(* CoDeSys 2.3 export: DACHA.EXP *)
(* Libraries: COMlibV2.lb6 25.2.14 08:37:08, ModbusRTU.lib 13.5.15 12:38:16, standard.lib 5.6.98 14:03:02, TcBABasic.lib 22.7.15 15:46:14, TcBase.lib 14.5.09 14:14:08, TcControllerToolbox.lib 19.6.15 13:33:48, TcFloatPC.lib 19.10.09 11:19:54, TcIoFunctions.lib 29.9.20 15:31:50, TcpIp.lib 6.5.15 09:25:52, TcSystem.lib 7.6.16 10:01:22, TcUtilities.lib 3.2.16 15:08:58 *)

(* Task configuration *)
TASK Standard (PRIORITY := 0, INTERVAL := T#2ms);
MAIN();
END_TASK
TASK main2 (PRIORITY := 1, INTERVAL := T#10ms);
MAIN2();
END_TASK

(* Global variable list: Global_Variables *)
VAR_GLOBAL


	Clear						: ClearComBuffer;
	MB							: ModbusRtuMaster_KL6x22B;
	TxBufferCom1				: ComBuffer;
	RxBufferCom1				: ComBuffer;
	SerialLineControlCom1			: SerialLineControl;
	ReceiveDataCom1			: ReceiveData;
	SendDataCom1				: SendData;


	Clear2						: ClearComBuffer;
	MB2							: ModbusRtuMaster_KL6x5B;
	TxBufferCom2				: ComBuffer;
	RxBufferCom2				: ComBuffer;
	SerialLineControlCom2			: SerialLineControl;
	ReceiveDataCom2			: ReceiveData;
	SendDataCom2				: SendData;
(*
	Clear3						: ClearComBuffer;
	MB3							: ModbusRtuMaster_KL6x22B;
	TxBufferCom3				: ComBuffer;
	RxBufferCom3				: ComBuffer;
	SerialLineControlCom3			: SerialLineControl;
	ReceiveDataCom3			: ReceiveData;
	SendDataCom3				: SendData;
*)

	Merc_address				: BYTE:=97;
	Sensor_CO2_high	 			: BYTE;	(*Старший байт датчика MH-Z19B*)
	Sensor_CO2_low 				: BYTE;	(*Младший байт датчика MH-Z19B*)
	iobroker						: iobroker_Struct;
	Modbus						: Modbus_Struct;
	Internal						: Internal_Struct;
	pwm_par_1f,pwm_par_2f		: ST_CTRL_PWM_OUT_PARAMS; (* настройки регулятора*)
	pwm_par_balkon				: ST_CTRL_PWM_OUT_PARAMS; (* настройки регулятора*)
	pwm_par_septik				: ST_CTRL_PWM_OUT_PARAMS; (* настройки регулятора*)
	pwm_par_sauna				: ST_CTRL_PWM_OUT_PARAMS; (* настройки регулятора*)
	pwm_par_fertA				: ST_CTRL_PWM_OUT_PARAMS; (* настройки регулятора*)
	pwm_par_fertB				: ST_CTRL_PWM_OUT_PARAMS; (* настройки регулятора*)

	pi_par_1f						: ST_CTRL_PI_PARAMS;			(*     *)
	pi_par_sauna					: ST_CTRL_PI_PARAMS;			(*     *)
	pi_par_fertA					: ST_CTRL_PI_PARAMS;			(*     *)
	pi_par_fertB					: ST_CTRL_PI_PARAMS;			(*     *)
	pi_par_balkon				: ST_CTRL_PI_PARAMS;			(*     *)

	Timer1					: TON;
	TimerRS485_2			: TON;
	TimerRS485_2Q			 :BOOL;

	TimerRS485_3			: TON;
	TimerRS485_3Q			 :BOOL;

	Timer1Q					: BOOL;
	Timer_day				:TON;
	Timer_dayQ				:BOOL;
	Timer_CO2				:TON;
(*	Timer_CO2Q				:BOOL; *)

	tmCheck					:TON;
	tmCheckQ				: BOOL;

	tmCheckE				:TON;
	tmCheckEQ				: BOOL;

	tmCheckM: TON;
(*
	MB_vars						: stMB;
	Mercury						: stMercury;
	iob_mqtt						: stIobroker;
*)
(*	Sensor_street_north_temp		: REAL;
	Sensor_sport_underfloor_temp	: REAL;
*)
	Sensor_control_temp			: WORD;
	Sensor_control_hum			: WORD;
(*	fert_pwm_levelA	: INT;
	fert_pwm_levelB	: INT;
*)
	Trigger_water_impulse_ponics	: F_TRIG;
	Trigger_A_impulse_ponics		: F_TRIG;
	Trigger_B_impulse_ponics		: F_TRIG;
	Trigger_water_impulse_teplica	: F_TRIG;
	Trigger_fertA_impulse_teplica	: F_TRIG;
	Trigger_fertB_impulse_teplica	: F_TRIG;
	Trigger_water_cnt_impulse_teplica	: F_TRIG;
	Poliv_liters				:	REAL;

	HW_teplica_pomp_fert_level			AT %Q*:BOOL;


(*Terminal 2*)
	HW_heat_first_floor					AT %QX0.0:BOOL;		(* Отопление 1 этаж *)
	HW_heat_second_floor				AT %QX0.1:BOOL;		(* Отопление 2 этаж *)
	HW_heat_sport						AT %QX0.2:BOOL;		(* Отопление спортзал *)
	HW_heat_underfloor					AT %QX0.3:BOOL;		(* Отопление подпол *)
	HW_heat_sauna						AT %QX0.4:BOOL;		(* Отопление сауна *)
	HW_heat_bathroom					AT %QX0.5:BOOL;		(* Отопление душевая *)
	HW_alarm							AT %QX0.6:BOOL;		(* Сирена *)
	HW_power_smoke_sen				AT %QX0.7:BOOL:=FALSE;		(* Питание датчиков дыма *)

(*Terminal 3*)
	HW_vorota							AT %QX1.0:BOOL;		(* Ворота *)
	HW_kalitka							AT %QX1.1:BOOL;		(* Калитка *)
	HW_pomp_house						AT %QX1.2:BOOL;		(* Насос водоснабжения дома *)
	HW_pomp_Garden					AT %QX1.3:BOOL;		(* Свободен*)
	HW_light_garden						AT %QX1.4:BOOL;		(* Прожектор двор *)
	HW_light_rassada						AT %QX1.5:BOOL;		(*Подсветка рассады на балконе *)
	HW_light_rezerv						AT %QX1.6:BOOL;		(* Резервное освещение *)
(*	HW_rezerv_term3_8					AT %QX1.7:BOOL; *)		(* Подогрев трубы в клубнике *)
	HW_poliv_flowers						AT %QX1.7:BOOL;

(*Terminal 4*)
	HW_vent_valve_input					AT %QX2.0:BOOL;		(* Клапан приточной вентиляции и Клапан вытяжной вентиляции *)
	HW_rezerv_term_4_3					AT %QX2.1:BOOL;		(*Свободен*)
	HW_trans_power						AT %QX2.2:BOOL;		(*Подача тока на трансформатор и реле ТЭН-а *)
	HW_vent_in_heat						AT %QX2.3:BOOL;		(* Подогрев притока - ТЭН *)
	HW_valve_pomp_teplica				AT %QX2.4:BOOL;		(* Клапан подачи воды в бочку теплицы*)
	HW_vent_in_trans_105_130				AT %QX2.5:BOOL:=FALSE;  (* Напряжение 110 или 130 В *)
	HW_vent_in_trans_160_220				AT %QX2.6:BOOL:=FALSE;  (* Напряжение 160 или 220 В *)
	HW_vent_in_trans_LO_HI				AT %QX2.7:BOOL:=FALSE;  (* Напряжение 110/130  или 160/220 В *)

(*Terminal 5*)
	HW_poliv_terrasa						AT %QX3.0:BOOL;		(* полив терраса  *)
	HW_poliv_zapad						AT %QX3.1:BOOL;		(* полив запад   *)
	HW_poliv_south						AT %QX3.2:BOOL;		(* полив юг   *)
	HW_poliv_north						AT %QX3.3:BOOL;		(* полив север   *)
	HW_septik_heat						AT %QX3.4:BOOL;		(*подогрев трубы до септика*)
	HW_power_supply_parnik				AT %QX3.5:BOOL;		(* Подача питания для механизма открывания окна*)
	HW_power_polarity_parnik				AT %QX3.6:BOOL;		(* Полярность питания для механизма открывания окна*)
	HW_parnik_heat						AT %QX3.7:BOOL;		(* подогрев трубы в парнике*)

(*Terminal 6*)
	HW_teplica_pomp_poliv				AT %Q*:BOOL; (*Teplica GR1.1*)
	HW_teplica_light						AT %Q*:BOOL; (*Teplica GR1.2*)
	HW_rezerv_6_3						AT %Q*:BOOL; (*Свободен*)
	HW_rezerv_6_4						AT %Q*:BOOL; (*Свободен*)
	HW_rezerv_6_5						AT %Q*:BOOL; (*Свободен*)
	HW_rezerv_6_6						AT %Q*:BOOL; (*Свободен*)
	HW_teplica_vent						AT %Q*:BOOL; (*Teplica GR1.7*)
	HW_teplica_heat						AT %Q*:BOOL; (*Teplica GR1.8*)




(*Terminal 7*)
	HW_rezerv_7_1						AT %Q*:BOOL;
	HW_rezerv_7_2						AT %Q*:BOOL;
	HW_rezerv_7_3						AT %Q*:BOOL;
	HW_ponics_pomp_water				AT %Q*:BOOL; (* 4 *)
	HW_ponics_pomp_tankA				AT %Q*:BOOL; (* 5 *)
	HW_ponics_pomp_tankB				AT %Q*:BOOL; (* 6 *)
	HW_ponics_pomp_main				AT %Q*:BOOL; (* 7 *)
	HW_balkon_heat						AT %Q*:BOOL; (* 8 *)

(*Terminal 8*)

(*	HW_teplica_pomp_fertA				AT %Q*:BOOL; (* PWM GND fert A*) (*Teplica GR2.1*)
	HW_teplica_pomp_fertB				AT %Q*:BOOL; (* PWM GND fert B*) (*Teplica GR2.2*)
*)
	fert_pwm_levelA						AT %Q*: UINT;
	fert_pwm_levelB						AT %Q*: UINT;
	pwm_ctrl_1							AT %Q*: USINT;
	pwm_ctrl_2							AT %Q*: USINT;


(*Terminal 9*)

	HW_PIR_terrasa						AT %IX56.0:BOOL;		(*PIR датчик терраса *)
	HW_PIR_zapad						AT %IX56.1:BOOL;		(*PIR датчик запад *)
	HW_PIR_vostok						AT %IX56.2:BOOL;		(*PIR датчик восток *)
	HW_PIR_sport						AT %IX56.3:BOOL;		(*PIR датчик спортзал *)
	HW_GERKON_drovnik					AT %IX56.4:BOOL;		(*Геркон дровник *)
	HW_GERKON_door					AT %IX56.5:BOOL;		(*Геркон дверь *)
	HW_sensor_smoke_1floor				AT %IX56.6:BOOL;		(*Датчик дыма 1 этаж *)
	HW_sensor_smoke_2floor				AT %IX56.7:BOOL;		(*Датчик дыма 2 этаж *)

(*Terminal 10*)
	HW_button_light_garden				AT %IX57.0:BOOL;		(* Кнопка прожектор терраса  *)
	HW_sensor_smoke_sport				AT %IX57.1:BOOL;		(*Датчик дыма спорт *)
	HW_button_vorota						AT %IX57.2:BOOL;		(* Кнопка открытия ворот  *)
	HW_rezerv_term_10_4					AT %IX57.3:BOOL;		(* Кнопка открытия калитки  *)
	HW_button_poliv_terrasa				AT %IX57.4:BOOL;		(* Кнопка полив терраса 2 часа  *)
	HW_button_poliv_zapad				AT %IX57.5:BOOL;		(* Кнопка полив запад  2 часа  *)
	HW_button_poliv_south				AT %IX57.6:BOOL;		(*  Кнопка полив юг  2 часа  *)
	HW_button_poliv_north					AT %IX57.7:BOOL;		(*  Кнопка полив север  2 часа  *)
(*Terminal 11*)
	HW_sensor_supply					AT %IX58.0:BOOL;		(* Датчик напряжения 220В  *)
	HW_GERKON_sklad					AT %IX58.1:BOOL;		(*Геркон склад*)
	HW_PIR_north_zapad					AT %IX58.2:BOOL;		(*PIR датчик  северо-запад*)
	HW_PIR_north_vostok					AT %IX58.3:BOOL;		(*PIR датчик  северо-восток*)

(*Terminal 12*)
	HW_vent_relay_pressure				 AT	%I*	:BOOL;		(*Реле давления вентиляции*)
	HW_sensor_smoke_stair				AT	%I*	:BOOL;		(*Датчик дыма лестница *)
	HW_sensor_smoke_3floor				AT	%I*	:BOOL;		(*Датчик дыма 3 этаж *)
	HW_sensor_smoke_drovnik			AT	%I*	:BOOL;		(*Датчик дыма дровник *)
	HW_sensor_smoke_sklad				AT	%I*	:BOOL;		(*Датчик дыма склад *)
	HW_button_alarm						AT	%I*	:BOOL;		(*Кнопка вкл и откл сирены *)
	HW_battery_low						 AT	%I*	:BOOL;		(*Датик низкого напряжения АКБ *)
	HW_water_tank_teplica_level			 AT	%I*	:BOOL;		(*Датчик уровня воды в бочке в теплице *) (*Teplica GR2.3*)

(*Terminal 13*)
	HW_water_tank_ponics_level_low		 AT	%I*	:BOOL;
	HW_water_tank_ponics_level_high		 AT	%I*	:BOOL;
	HW_sensor_fluid_alarm				 AT	%I*	:BOOL;
	HW_water_counter					 AT	%I*	:BOOL;
	HW_I_rez5							 AT	%I*	:BOOL;
	HW_I_rez6							 AT	%I*	:BOOL;
	HW_I_rez7							 AT	%I*	:BOOL;
	HW_I_rez8							 AT	%I*	:BOOL;

(*Terminal 14*)
	HW_impulse_water_teplica				 AT	%I*	:BOOL; (*Teplica GR2.4*)
	HW_impulse_fertA_teplica				 AT	%I*	:BOOL; (*Teplica GR2.5*)
	HW_impulse_fertB_teplica				 AT	%I*	:BOOL; (*Teplica GR2.6*)
	HW_impulse_water_ponics				 AT	%I*	:BOOL;

	HW_impulse_tankA_ponics				 AT	%I*	:BOOL;
	HW_impulse_tankB_ponics				 AT	%I*	:BOOL;
	HW_I_rez15							 AT	%I*	:BOOL;
	HW_I_rez16							 AT	%I*	:BOOL;

(*Terminal 15*)
	HW_temp_first_floor					AT %IW40:INT;	(* Датчик температуры 1 этаж *)
	HW_temp_second_floor				AT %IW42:INT;	(* Датчик температуры 2 этаж *)
	HW_temp_sauna						AT %IW44:INT;	(* Датчик температуры сауна*)
	HW_temp_sport						AT %IW46:INT;	(* Датчик температуры спортзал *)

(*Terminal 16*)
	HW_temp_underfloor					AT %IW48:INT;	(* Датчик температуры подпол *)
	HW_temp_balkon						AT %IW50:INT;	(* Датчик температуры  *)
	HW_temp_street						AT %IW52:INT;	(* Датчик температуры улица *)
	HW_temp_vent						AT %IW54:INT;	(* Датчик температуры притока вентиляции *)



END_VAR

(* Global variable list: TwinCAT_Configuration *)
(* Generated automatically by TwinCAT - (read only) *)
VAR_CONFIG
	MAIN2.ToFromNovRam AT %QB584 : DataToFromNovram;	(*  ~ {LinkedWith:TIID^Device 2 (NOV/DP-RAM)^Outputs^Var 403} *)
	.MB.InData AT %IB68 : MB_KL6inData22B;
	.MB.OutData AT %QB376 : MB_KL6outData22B;
	.MB2.InData AT %IB96 : MB_KL6inData5B;
	.MB2.OutData AT %QB344 : MB_KL6outData5B;
	.HW_teplica_pomp_fert_level AT %QX476.0 : BOOL;
	.HW_teplica_pomp_poliv AT %QX480.3 : BOOL;	(*  ~ {LinkedWith:TIID^Device 1 (CX9000-KBus)^CX9000-KB^Term 6 (KL2408)^Channel 1^Output} *)
	.HW_teplica_light AT %QX480.2 : BOOL;	(*  ~ {LinkedWith:TIID^Device 1 (CX9000-KBus)^CX9000-KB^Term 6 (KL2408)^Channel 2^Output} *)
	.HW_rezerv_6_3 AT %QX724.0 : BOOL;	(*  ~ {LinkedWith:TIID^Device 1 (CX9000-KBus)^CX9000-KB^Term 6 (KL2408)^Channel 3^Output} *)
	.HW_rezerv_6_4 AT %QX724.1 : BOOL;	(*  ~ {LinkedWith:TIID^Device 1 (CX9000-KBus)^CX9000-KB^Term 6 (KL2408)^Channel 4^Output} *)
	.HW_rezerv_6_5 AT %QX724.2 : BOOL;	(*  ~ {LinkedWith:TIID^Device 1 (CX9000-KBus)^CX9000-KB^Term 6 (KL2408)^Channel 5^Output} *)
	.HW_rezerv_6_6 AT %QX724.3 : BOOL;	(*  ~ {LinkedWith:TIID^Device 1 (CX9000-KBus)^CX9000-KB^Term 6 (KL2408)^Channel 6^Output} *)
	.HW_teplica_vent AT %QX480.0 : BOOL;	(*  ~ {LinkedWith:TIID^Device 1 (CX9000-KBus)^CX9000-KB^Term 6 (KL2408)^Channel 7^Output} *)
	.HW_teplica_heat AT %QX480.1 : BOOL;	(*  ~ {LinkedWith:TIID^Device 1 (CX9000-KBus)^CX9000-KB^Term 6 (KL2408)^Channel 8^Output} *)
	.HW_rezerv_7_1 AT %QX724.4 : BOOL;	(*  ~ {LinkedWith:TIID^Device 1 (CX9000-KBus)^CX9000-KB^Term 7 (KL2408)^Channel 1^Output} *)
	.HW_rezerv_7_2 AT %QX724.5 : BOOL;	(*  ~ {LinkedWith:TIID^Device 1 (CX9000-KBus)^CX9000-KB^Term 7 (KL2408)^Channel 2^Output} *)
	.HW_rezerv_7_3 AT %QX724.6 : BOOL;	(*  ~ {LinkedWith:TIID^Device 1 (CX9000-KBus)^CX9000-KB^Term 7 (KL2408)^Channel 3^Output} *)
	.HW_ponics_pomp_water AT %QX484.2 : BOOL;	(*  ~ {LinkedWith:TIID^Device 1 (CX9000-KBus)^CX9000-KB^Term 7 (KL2408)^Channel 4^Output} *)
	.HW_ponics_pomp_tankA AT %QX484.3 : BOOL;	(*  ~ {LinkedWith:TIID^Device 1 (CX9000-KBus)^CX9000-KB^Term 7 (KL2408)^Channel 5^Output} *)
	.HW_ponics_pomp_tankB AT %QX484.4 : BOOL;	(*  ~ {LinkedWith:TIID^Device 1 (CX9000-KBus)^CX9000-KB^Term 7 (KL2408)^Channel 6^Output} *)
	.HW_ponics_pomp_main AT %QX484.1 : BOOL;	(*  ~ {LinkedWith:TIID^Device 1 (CX9000-KBus)^CX9000-KB^Term 7 (KL2408)^Channel 7^Output} *)
	.HW_balkon_heat AT %QX580.0 : BOOL;	(*  ~ {LinkedWith:TIID^Device 1 (CX9000-KBus)^CX9000-KB^Term 7 (KL2408)^Channel 8^Output} *)
	.fert_pwm_levelA AT %QB708 : UINT;	(*  ~ {LinkedWith:TIID^Device 1 (CX9000-KBus)^CX9000-KB^Term 8 (KL2502)^Channel 1^Data Out} *)
	.fert_pwm_levelB AT %QB710 : UINT;	(*  ~ {LinkedWith:TIID^Device 1 (CX9000-KBus)^CX9000-KB^Term 8 (KL2502)^Channel 2^Data Out} *)
	.pwm_ctrl_1 AT %QB712 : USINT;	(*  ~ {LinkedWith:TIID^Device 1 (CX9000-KBus)^CX9000-KB^Term 8 (KL2502)^Channel 1^Ctrl} *)
	.pwm_ctrl_2 AT %QB713 : USINT;	(*  ~ {LinkedWith:TIID^Device 1 (CX9000-KBus)^CX9000-KB^Term 8 (KL2502)^Channel 2^Ctrl} *)
	.HW_vent_relay_pressure AT %IX104.0 : BOOL;	(*  ~ {LinkedWith:TIID^Device 1 (CX9000-KBus)^CX9000-KB^Term 12 (KL1408)^Channel 1^Input} *)
	.HW_sensor_smoke_stair AT %IX140.0 : BOOL;	(*  ~ {LinkedWith:TIID^Device 1 (CX9000-KBus)^CX9000-KB^Term 12 (KL1408)^Channel 2^Input} *)
	.HW_sensor_smoke_3floor AT %IX132.1 : BOOL;	(*  ~ {LinkedWith:TIID^Device 1 (CX9000-KBus)^CX9000-KB^Term 12 (KL1408)^Channel 3^Input} *)
	.HW_sensor_smoke_drovnik AT %IX132.2 : BOOL;	(*  ~ {LinkedWith:TIID^Device 1 (CX9000-KBus)^CX9000-KB^Term 12 (KL1408)^Channel 4^Input} *)
	.HW_sensor_smoke_sklad AT %IX132.3 : BOOL;	(*  ~ {LinkedWith:TIID^Device 1 (CX9000-KBus)^CX9000-KB^Term 12 (KL1408)^Channel 5^Input} *)
	.HW_button_alarm AT %IX136.0 : BOOL;	(*  ~ {LinkedWith:TIID^Device 1 (CX9000-KBus)^CX9000-KB^Term 12 (KL1408)^Channel 6^Input} *)
	.HW_battery_low AT %IX132.0 : BOOL;	(*  ~ {LinkedWith:TIID^Device 1 (CX9000-KBus)^CX9000-KB^Term 12 (KL1408)^Channel 7^Input} *)
	.HW_water_tank_teplica_level AT %IX144.0 : BOOL;	(*  ~ {LinkedWith:TIID^Device 1 (CX9000-KBus)^CX9000-KB^Term 12 (KL1408)^Channel 8^Input} *)
	.HW_water_tank_ponics_level_low AT %IX168.0 : BOOL;	(*  ~ {LinkedWith:TIID^Device 1 (CX9000-KBus)^CX9000-KB^Term 13 (KL1408)^Channel 1^Input} *)
	.HW_water_tank_ponics_level_high AT %IX168.1 : BOOL;	(*  ~ {LinkedWith:TIID^Device 1 (CX9000-KBus)^CX9000-KB^Term 13 (KL1408)^Channel 2^Input} *)
	.HW_sensor_fluid_alarm AT %IX164.0 : BOOL;	(*  ~ {LinkedWith:TIID^Device 1 (CX9000-KBus)^CX9000-KB^Term 13 (KL1408)^Channel 3^Input} *)
	.HW_water_counter AT %IX164.1 : BOOL;	(*  ~ {LinkedWith:TIID^Device 1 (CX9000-KBus)^CX9000-KB^Term 13 (KL1408)^Channel 4^Input} *)
	.HW_I_rez5 AT %IX148.4 : BOOL;	(*  ~ {LinkedWith:TIID^Device 1 (CX9000-KBus)^CX9000-KB^Term 13 (KL1408)^Channel 5^Input} *)
	.HW_I_rez6 AT %IX148.5 : BOOL;	(*  ~ {LinkedWith:TIID^Device 1 (CX9000-KBus)^CX9000-KB^Term 13 (KL1408)^Channel 6^Input} *)
	.HW_I_rez7 AT %IX148.6 : BOOL;	(*  ~ {LinkedWith:TIID^Device 1 (CX9000-KBus)^CX9000-KB^Term 13 (KL1408)^Channel 7^Input} *)
	.HW_I_rez8 AT %IX148.7 : BOOL;	(*  ~ {LinkedWith:TIID^Device 1 (CX9000-KBus)^CX9000-KB^Term 13 (KL1408)^Channel 8^Input} *)
	.HW_impulse_water_teplica AT %IX152.0 : BOOL;	(*  ~ {LinkedWith:TIID^Device 1 (CX9000-KBus)^CX9000-KB^Term 14 (KL1408)^Channel 1^Input} *)
	.HW_impulse_fertA_teplica AT %IX152.1 : BOOL;	(*  ~ {LinkedWith:TIID^Device 1 (CX9000-KBus)^CX9000-KB^Term 14 (KL1408)^Channel 2^Input} *)
	.HW_impulse_fertB_teplica AT %IX152.2 : BOOL;	(*  ~ {LinkedWith:TIID^Device 1 (CX9000-KBus)^CX9000-KB^Term 14 (KL1408)^Channel 3^Input} *)
	.HW_impulse_water_ponics AT %IX156.0 : BOOL;	(*  ~ {LinkedWith:TIID^Device 1 (CX9000-KBus)^CX9000-KB^Term 14 (KL1408)^Channel 4^Input} *)
	.HW_impulse_tankA_ponics AT %IX156.1 : BOOL;	(*  ~ {LinkedWith:TIID^Device 1 (CX9000-KBus)^CX9000-KB^Term 14 (KL1408)^Channel 5^Input} *)
	.HW_impulse_tankB_ponics AT %IX156.2 : BOOL;	(*  ~ {LinkedWith:TIID^Device 1 (CX9000-KBus)^CX9000-KB^Term 14 (KL1408)^Channel 6^Input} *)
	.HW_I_rez15 AT %IX149.6 : BOOL;	(*  ~ {LinkedWith:TIID^Device 1 (CX9000-KBus)^CX9000-KB^Term 14 (KL1408)^Channel 7^Input} *)
	.HW_I_rez16 AT %IX149.7 : BOOL;	(*  ~ {LinkedWith:TIID^Device 1 (CX9000-KBus)^CX9000-KB^Term 14 (KL1408)^Channel 8^Input} *)
END_VAR

(* Data type *)
TYPE DataToFromNovram :
STRUCT

	Target_CO2_mem					:		INT:=600;
	First_floor_temp_target_mem		:		INT:=5;
	Second_floor_temp_target_mem		:		INT:=5;
	Sport_temp_target_mem			:		INT:=5;
	Sauna_temp_target_mem			:		INT:=5;
	Underfloor_temp_target_mem		:		INT:=5;
	Underfloor_humidity_target_mem	:		INT:=90;

	Pomp_house_mem				:		BOOL:=FALSE;
	Pomp_garden_mem				:		BOOL:=FALSE;

	Light_garden_mem				:		BOOL:=FALSE;

	Vent_mem						:		BOOL:=FALSE;
	Vent_heat_mem					:		INT;
	Vent_heat_level_mem				:		BOOL;

	Poliv_zapad_minutes				:		INT:=90;
	Poliv_terrasa_minutes				:		INT:=90;
	Poliv_south_minutes				:		INT:=90;
	Poliv_north_minutes				:		INT:=90;

	Teplica_temp_set_high			:	INT:=21;
	Teplica_temp_set_low				:	INT:=18;
	Teplica_light_set_low				:	INT:=4000;
	Teplica_light_allow				:	BOOL;
	Teplica_poliv_kf					:	INT:=1025;
	Teplica_fertA_kf					:	INT:=11450;
	Teplica_fertB_kf					:	INT:=11450;

	Teplica_set_poliv					:	REAL;
	Teplica_set_fertA					:	REAL;
	Teplica_set_fertB					:	REAL;
	Teplica_set_max_poliv_time		:	UDINT;
	Teplica_set_max_fertA_time		:	UDINT;
	Teplica_set_max_fertB_time		:	UDINT;
	Teplica_set_clear_time			:	UDINT:=5;

	Teplica_set_temp_pomp_cold		:	INT:=24;
	Teplica_set_temp_window_open	:	INT:=21;
	Teplica_set_poliv_before_fert		:	INT:=50;

	Teplica_set_temp_tank			:	INT:=-60;
	Teplica_fert_kf					:	INT:=12;
	Teplica_zone_poliv				:	BOOL;
	Teplica_type_fert					:	BOOL;
	Teplica_type_poliv				:	BOOL;
	Teplica_set_finish_clear_time		:	INT:=5;
	Teplica_set_finish_clear_vol		:	INT:=1;

	Ponics_start_mintutes_poliv			:	INT:=0;
	Ponics_start_minutes_doliv_AB		:	INT:=30;
	Ponics_start_minutes_doliv_water	:	INT:=20;
	Ponics_set_doliv_AB				:	REAL:=0.1;
	Ponics_set_doliv_water			:	REAL:=3;
	Ponics_set_max_poliv_time			:	INT:=3000;
	Ponics_set_max_doliv_A_time		:	INT:=30;
	Ponics_set_max_doliv_water_time	:	INT:=600;
	Ponics_set_EC					:	REAL:=2.0;
	Balkon_set_temp					:	INT:=21;
	Ponics_A_kf						:	INT:=7030;
	Ponics_B_kf						:	INT:=7030;
	Ponics_water_kf					:	INT:=7030;

	Sensor_house_water_imp			:	UDINT;
	Parnik_temp_step1_window			:	INT:=18;
	Parnik_temp_step2_window			:	INT:=24;
	Parnik_set_auto_window			:	BOOL;
	Parnik_current_level_window		:	INT;
	Parnik_manual_level_window		:	INT;



END_STRUCT
END_TYPE

(* Data type *)
TYPE DataToFromNovram2 :
STRUCT

	Target_CO2_mem					:		INT;
	First_floor_temp_target_mem		:		INT;
	Second_floor_temp_target_mem		:		INT;
	Sport_temp_target_mem			:		INT;
	Sauna_temp_target_mem			:		INT;
	Underfloor_temp_target_mem		:		INT;
	Underfloor_humidity_target_mem	:		INT;

	Pomp_house_mem				:		BOOL;
	Pomp_garden_mem				:		BOOL;

	Light_garden_mem				:		BOOL;

	Vent_mem						:		BOOL;
	Vent_heat_mem					:		INT;
	Vent_heat_level_mem				:		BOOL;

	Poliv_zapad_minutes				:		INT;
	Poliv_terrasa_minutes				:		INT;
	Poliv_south_minutes				:		INT;
	Poliv_north_minutes				:		INT;

	Teplica_temp_set_high			:	INT;
	Teplica_temp_set_low				:	INT;
	Teplica_light_set_low				:	INT;
	Teplica_light_allow				:	BOOL;
	Teplica_poliv_kf					:	INT;
	Teplica_fertA_kf					:	INT;
	Teplica_fertB_kf					:	INT;

	Teplica_set_poliv					:	REAL;
	Teplica_set_fertA					:	REAL;
	Teplica_set_fertB					:	REAL;
	Teplica_set_max_poliv_time		:	UDINT;
	Teplica_set_max_fertA_time		:	UDINT;
	Teplica_set_max_fertB_time		:	UDINT;
	Teplica_set_clear_time			:	UDINT;

END_STRUCT
END_TYPE

(* Data type *)
TYPE Internal_struct :
STRUCT
	Drovnik_temp					 :	REAL; 	(*12382*)			(* PT1000 *)
	Sklad_temp					 :	REAL; 	(*12384*)			(* PT1000 *)
	Rezerv_temp					 :	REAL; 	(*12386*)			(* PT1000 *)

	First_floor_temp 				:	REAL;	(*12288+100=12388*) (* PT1000 *)
	First_floor_hum 				:	REAL;	(*12390*)			(*SHT20		#1*)
	First_floor_CO2				:	REAL;	(*12392*)
	First_floor_temp_SHT30		:	REAL;	(*12394*)			(*SHT20		#1*)

	Second_floor_hum			:	REAL;	(*12396*)			(*SHT20		#2*)
	Second_floor_temp 			:	REAL;	(*12398*) 		(* PT1000 *)
	Second_floor_CO2 			:	REAL;	(*12400*)
	Sport_temp	 				:	REAL;	(*12402*)			(* PT1000 *)

	Sauna_temp	 				:	REAL;	(*12404*)			(* PT1000 *)
	Underfloor_temp				:	REAL;	(*12406*)			(* PT1000 *)
	Underfloor_hum				:	REAL;	(*12408*)			(*SHT20		#3*)
	Sport_underfloor_temp			:	REAL;	(*12410*)			(* PT1000 *)

	Sport_underfloor_hum			:	REAL;	(*12412*)			(*SHT20		#4*)
	Street_temp					:	REAL;	(*12414*)			(* PT1000 *)
	Vent_temp					:	REAL;	(*12416*)			(* PT1000 *)
	Sklad_temp_SHT20			:	REAL;	(*12418*)			(*SHT20		#5*)
	Sklad_hum					:	REAL;	(*12420*)			(*SHT20		#5*)
	Temp_vent_in				:	REAL;	(*12422*)			(* unused *)

	Sport_temp_SHT30			:	REAL;	(*12458 *)		(*SHT20		#6*)
	Sport_hum					:	REAL;	(*12460 *)		(*SHT20		#6*)
	Drovnik_temp_SHT30			:	REAL;	(*12462 *)		(*SHT20		#6*)
	Drovnik_hum					:	REAL;	(*12464 *)		(*SHT20		#6*)


	Uv1							:	REAL;	(*12424*)
	Uv2							:	REAL;	(*12426*)
	Uv3							:	REAL;	(*12428*)
	Pw1							:	REAL;	(*12430*)
	Pw2							:	REAL;	(*12432*)
	Pw3							:	REAL;	(*12434*)
	Pw_total						:	REAL;	(*12436*)
	Ia1							:	REAL;	(*12438*)
	Ia2							:	REAL;	(*12440*)
	Ia3							:	REAL;	(*12442*)
	E_T1						:	REAL;	(*12444*)
	E_T2						:	REAL; 	(*12288+158=12446*)

	Second_floor_temp_SHT30			:	REAL;	(*12448 *)		(*SHT20		#2*)
	Underfloor_temp_SHT30			:	REAL;	(*12450 *)		(*SHT20		#3*)
	Sport_underfloor_temp_SHT30		:	REAL;	(*12452 *)		(*SHT20		#4*)
	Street_temp_SHT20				:	REAL;	(*12454 *)		(*SHT20		#6*)
	Street_hum						:	REAL;	(*12456 *)		(*SHT20		#6*)

	Teplica_temp_SHT30				:	REAL;	(**)
	Teplica_hum_SHT30				:	REAL;	(**)


END_STRUCT
END_TYPE

(* Data type *)
TYPE iobroker_Struct  :
STRUCT
(*	Vent_status				: 	INT;
	Valve_status				: 	INT;
	First_floor_temp 			:	REAL;
	First_floor_temp_target 		:	INT;
	First_floor_hum 			:	REAL;
	First_floor_CO2			:	REAL;
	Kitchen_room_temp		:	REAL;
	Kitchen_room_hum		:	REAL;
	Second_floor_temp 		:	REAL;
	Second_floor_temp_target 	:	INT;
	Second_floor_CO2 		:	REAL;
	Sport_temp	 			:	REAL;
	Sport_temp_target			:	INT;
	Sauna_temp	 			:	REAL;
	Sauna_temp_target		:	INT;
	Underfloor_temp			:	REAL;
	Underfloor_temp_target	:	INT;
	Underfloor_humidity		:	REAL;
	Underfloor_humidity_target	:	INT;
	Sport_underfloor_temp		:	REAL;
	Sport_underfloor_hum		:	REAL;
	Street_temp				:	REAL;
	Vent_temp				:	REAL;
	Street_north_temp			:	REAL;
	Street_north_hum			:	REAL;
*)
	PIR_terrasa				:	BOOL:=TRUE;
	PIR_zapad				:	BOOL:=TRUE;
	PIR_vostok				:	BOOL:=TRUE;
	PIR_sport				:	BOOL:=TRUE;
	GERKON_drovnik			:	BOOL:=TRUE;
	Smoke					:	BOOL;
	Button_light_garden		:	BOOL;
	Light_garden				:	BOOL;
	Vorota_active				:	BOOL:=FALSE;
	Vorota_open_active		:	BOOL:=FALSE;
(*	Poliv_zapad				:	BOOL;
	Poliv_terrasa				:	BOOL;
	Poliv_south				:	BOOL;
	Poliv_north				:	BOOL;
*)
(*
	Vent_input_level			:	INT;  (*  0-220 V  *)
	Vent_output_level			:	INT; (*0-100%*)
	Temp_vent_in			:	REAL;
	Vent_valve_status			:	INT;
	Security_status			:	BOOL;
	Target_CO2				:	INT;
	Vent						:	BOOL;
	Vent_underfloor			:	BOOL;
	Vent_out					:	BOOL;
	Vent_heat				:	INT;
	Vent_heat_level			:	BOOL;
	Vorota					:	BOOL;
	Vorota_open				:	BOOL;
	Kalitka					:	BOOL;
	
	Sensor_supply			:	BOOL;
	Pomp_house				:	BOOL;
	Pomp_garden			:	BOOL;
	Light_garden				:	BOOL;
	Poliv_zapad				:	BOOL;
	Poliv_terrasa				:	BOOL;
	Poliv_south				:	BOOL;
	Poliv_zapad_minutes		:	INT;
	Poliv_terrasa_minutes		:	INT;
	Poliv_south_minutes		:	INT;
	Uv1						:	REAL;
	Uv2						:	REAL;
	Uv3						:	REAL;
	Pw1						:	REAL;
	Pw2						:	REAL;
	Pw3						:	REAL;
	Pw_total					:	REAL;
	Ia1						:	REAL;
	Ia2						:	REAL;
	Ia3						:	REAL;
	E_T1					:	REAL;
	E_T2					:	REAL; (* 64 values*)
*)

(*	M1T1					:	DWORD:=0;
	M1T2					:	DWORD:=0; (* 66 values*)

	M2T1					:	DWORD:=0; (* 67 values*)
	M2T2					:	DWORD:=0;
	M3T1					:	DWORD:=0;
	M3T2					:	DWORD:=0;
	M4T1					:	DWORD:=0; (* 70 values*)
	M4T2					:	DWORD:=0;
	M5T1					:	DWORD:=0;
	M5T2					:	DWORD:=0;
	M6T1					:	DWORD:=0;
	M6T2					:	DWORD:=0;
	M7T1					:	DWORD:=0;
	M7T2					:	DWORD:=0;
	M8T1					:	DWORD:=0;
	M8T2					:	DWORD:=0;
	M9T1					:	DWORD:=0;
	M9T2					:	DWORD:=0;
	M10T1					:	DWORD:=0;
	M10T2					:	DWORD:=0;
	M11T1					:	DWORD:=0;
	M11T2					:	DWORD:=0;
	M12T1					:	DWORD:=0;
	M12T2					:	DWORD:=0;   (* 86 values*)
*)

END_STRUCT
END_TYPE

(* Data type *)
TYPE Modbus_struct :
STRUCT

	M1T1							AT %MW0	:REAL;  	(* modbus address 12288 *)
	M1T2							AT %MW4	:REAL;	(* 12290 *)
	M2T1							AT %MW8	:REAL;	(* 12292 *)
	M2T2							AT %MW12	:REAL;	 (* 12294 *)
	M3T1							AT %MW16	:REAL;	 (* 12296 *)
	M3T2							AT %MW20	:REAL;	 (* 12298 *)
	M4T1							AT %MW24	:REAL;	 (* 12300 *)
	M4T2							AT %MW28	:REAL;	 (* 12302 *)
	M5T1							AT %MW32	:REAL;	 (* 12304 *)
	M5T2							AT %MW36	:REAL;	 (* 12306 *)
	M6T1							AT %MW40	:REAL;	 (* 12308 *)
	M6T2							AT %MW44	:REAL;	(* 12310 *)
	M7T1							AT %MW48	:REAL;	 (* 12312 *)
	M7T2							AT %MW52	:REAL;	 (* 12314 *)
	M8T1							AT %MW56	:REAL;	 (* 12316 *)
	M8T2							AT %MW60	:REAL;	(* 12318 *)
	M9T1							AT %MW64	:REAL;	(* 12320 *)
	M9T2							AT %MW68	:REAL;	(* 12322 *)
	M10T1							AT %MW72	:REAL;	(* 12324 *)
	M10T2							AT %MW76	:REAL;	(* 12326 *)
	M11T1							AT %MW80	:REAL;	(* 12328 *)
	M11T2							AT %MW84	:REAL;	(* 12330 *)
	M12T1							AT %MW88	:REAL;	(* 12332 *)
	M12T2							AT %MW92	:REAL;	(* 12334 *)


	Vent_status					AT %MB100	:	INT;		(*12288+50=12338*)
	Valve_status					AT %MB102	: 	INT;		(*12339*)
	First_floor_temp_target 			AT %MB104	:	INT:=5;		(*12340*)
	Second_floor_temp_target 		AT %MB106	:	INT:=5;		(*12341*)
	Sport_temp_target				AT %MB108	:	INT:=5;		(*12342*)
	Sauna_temp_target			AT %MB110	:	INT:=0;		(*12343*)
	Underfloor_temp_target		AT %MB112	:	INT:=5;		(*12344*)
	Underfloor_humidity_target		AT %MB114	:	INT:=90;		(*12345*)
	PIR_terrasa					AT %MB116	:	BOOL:=TRUE;	(*12346*)
	PIR_zapad					AT %MB118	:	BOOL:=TRUE;	(*12347*)
	PIR_vostok					AT %MB120	:	BOOL:=TRUE;	(*12348*)
	PIR_sport					AT %MB122	:	BOOL:=TRUE;	(*12349*)
	GERKON_drovnik				AT %MB124	:	BOOL:=TRUE;	(*12288+62=12350*)

	Vent_input_level				AT %MB126	:	INT; 			 (*12351			*  0-220 V  *)
	Vent_output_level				AT %MB128	:	INT; 			(*12352			0-100%*)
	Vent_valve_status				AT %MB130	:	INT;		(*12353*)
	Target_CO2					AT %MB132	:	INT:=600;		(*12354*)
	Security_status				AT %MB134	:	BOOL;	(*12355*)
	Vent							AT %MB136	:	BOOL;	(*12356*)
	Vent_underfloor				AT %MB138	:	BOOL;	(*12357*)
	Vent_out						AT %MB140	:	BOOL;	(*12358*)
	Vent_heat					AT %MB142	:	INT:=1;		(*12359*)
	Vent_heat_level				AT %MB144	:	BOOL;	(*12360*)
	Vorota						AT %MB146	:	BOOL;	(*12361*)
	Vorota_open					AT %MB148	:	BOOL;	(*12362*)
	Kalitka						AT %MB150	:	BOOL;	(*12363*)
(*
	Smoke						AT %MB152	:	BOOL;	(*12364*)
*)
	Sensor_supply				AT %MB154	:	BOOL;	(*12365*)
	Pomp_house					AT %MB156	:	BOOL;	(*12366*)
	Pomp_garden				AT %MB158	:	BOOL;	(*12367*)
	Light_garden					AT %MB160	:	BOOL;	(*12368*)
	Poliv_zapad					AT %MB162	:	BOOL;	(*12369*)
	Poliv_terrasa					AT %MB164	:	BOOL;	(*12370*)
	Poliv_south					AT %MB166	:	BOOL;	(*12371*)
	Poliv_zapad_minutes			AT %MB168	:	INT:=60;		(*12372*)
	Poliv_terrasa_minutes			AT %MB170	:	INT:=60;		(*12373*)
	Poliv_south_minutes			AT %MB172	:	INT:=60;		(*12288 +86=  12374*)
	Poliv_north_minutes			AT %MB174	:	INT:=60	;	(*12375 *)
	Poliv_north					AT %MB176	:	BOOL;	(*12376*)
	Poliv_flowers					AT %MB178	:	BOOL;	(*12377*)
	Poliv_flowers_minutes			AT %MB180	:	INT:=60	;	(*12378 *)
	Poliv_flowers_minutes_est		AT %MB182	:	INT;		(*12379 *)







	Drovnik_temp					AT %MW188 :	REAL; 	(*12382*)			(* PT1000 *)
	Sklad_temp					AT %MW192 :	REAL; 	(*12384*)			(* PT1000 *)
	Rezerv_temp					AT %MW196 :	REAL; 	(*12386*)			(* PT1000 *)

	First_floor_temp 				AT %MW200	:	REAL;	(*12288+100=12388*) (* PT1000 *)
	First_floor_hum 				AT %MW204	:	REAL;	(*12390*)			(*SHT20		#1*)
	First_floor_CO2				AT %MW208	:	REAL;	(*12392*)
	First_floor_temp_SHT30		AT %MW212	:	REAL;	(*12394*)			(*SHT20		#1*)

	Second_floor_hum			AT %MW216	:	REAL;	(*12396*)			(*SHT20		#2*)
	Second_floor_temp 			AT %MW220	:	REAL;	(*12398*) 		(* PT1000 *)
	Second_floor_CO2 			AT %MW224	:	REAL;	(*12400*)
	Sport_temp	 				AT %MW228	:	REAL;	(*12402*)			(* PT1000 *)

	Sauna_temp	 				AT %MW232	:	REAL;	(*12404*)			(* PT1000 *)
	Underfloor_temp				AT %MW236	:	REAL;	(*12406*)			(* PT1000 *)
	Underfloor_hum				AT %MW240	:	REAL;	(*12408*)			(*SHT20		#3*)
	Sport_underfloor_temp			AT %MW244	:	REAL;	(*12410*)			(* PT1000 *)

	Sport_underfloor_hum			AT %MW248	:	REAL;	(*12412*)			(*SHT20		#4*)
	Street_temp					AT %MW252	:	REAL;	(*12414*)			(* PT1000 *)
	Vent_temp					AT %MW256	:	REAL;	(*12416*)			(* PT1000 *)
	Sklad_temp_SHT20			AT %MW260	:	REAL;	(*12418*)			(*SHT20		#5*)
	Sklad_hum					AT %MW264	:	REAL;	(*12420*)			(*SHT20		#5*)
	Temp_vent_in				AT %MW268	:	REAL;	(*12422*)			(* unused *)


	Uv1							AT %MW272	:	REAL;	(*12424*)
	Uv2							AT %MW276	:	REAL;	(*12426*)
	Uv3							AT %MW280	:	REAL;	(*12428*)
	Pw1							AT %MW284	:	REAL;	(*12430*)
	Pw2							AT %MW288	:	REAL;	(*12432*)
	Pw3							AT %MW292	:	REAL;	(*12434*)
	Pw_total						AT %MW296	:	REAL;	(*12436*)
	Ia1							AT %MW300	:	REAL;	(*12438*)
	Ia2							AT %MW304	:	REAL;	(*12440*)
	Ia3							AT %MW308	:	REAL;	(*12442*)
	E_T1						AT %MW312	:	REAL;	(*12444*)
	E_T2						AT %MW316	:	REAL; 	(*12288+158=12446*)

	Second_floor_temp_SHT30		AT %MW320	:	REAL;	(*12448 *)		(*SHT20		#2*)
	Underfloor_temp_SHT30		AT %MW324	:	REAL;	(*12450 *)		(*SHT20		#3*)
	Sport_underfloor_temp_SHT30	AT %MW328	:	REAL;	(*12452 *)		(*SHT20		#4*)
	Street_temp_SHT20			AT %MW332	:	REAL;	(*12454 *)		(*SHT20		#6*)
	Street_hum					AT %MW336	:	REAL;	(*12456 *)		(*SHT20		#6*)
	Sport_temp_SHT30			AT %MW340	:	REAL;	(*12458 *)		(*SHT20		#6*)
	Sport_hum					AT %MW344	:	REAL;	(*12460 *)		(*SHT20		#6*)
	Drovnik_temp_SHT30			AT %MW348	:	REAL;	(*12462 *)		(*SHT20		#6*)
	Drovnik_hum					AT %MW352	:	REAL;	(*12464 *)		(*SHT20		#6*)

	Teplica_window_opener		AT  %MB356	:	BOOL;	(*12288+178=12466*)
	Teplica_pomp_cold				AT %MB358	:	BOOL;	(*12467*)
	Teplica_set_temp_pomp_cold		AT %MB360	:	INT:=32;	(*12468*)
	Teplica_set_temp_window_open	AT %MB362	:	INT:=23;	(*12469*)
	Teplica_set_poliv_before_fert		AT %MB364	:	INT:=10;	(*12470*)
	Teplica_pomp_fert_level			AT %MB366	:	BOOL;	(*12471*)

	Poliv_valve_winter					AT %MB368	:	BOOL;	(*12472*)
	Heat_pipe_water_winter			AT %MB370	:	BOOL;	(*12473*)
	Heat_pipe_septik_winter			AT %MB372	:	BOOL;	(*12474*)

(* PONIC old1
	Ponics_impulse_water_cnt		AT  %MW368	:	UDINT;	(*12472*)
	Ponics_impulse_A_cnt			AT  %MW372	:	UDINT;	(*12474*)
	Ponics_impulse_B_cnt			AT  %MW376	:	UDINT;	(*12476*)

	Ponics_set_max_poliv_time			AT  %MB380	:	UINT;	(*12478*)
	Ponics_set_max_doliv_water_time	AT  %MB382	:	UINT;	(*12479*)
	Ponics_set_max_doliv_A_time		AT  %MB384	:	UINT;	(*12480*)
	Ponics_set_max_doliv_B_time		AT  %MB386	:	UINT;	(*12481*)
	Ponics_poliv_active				AT  %MB388	:	BOOL;	(*12482*)
	Ponics_poliv_break				AT  %MB390	:	BOOL;	(*12483*)
	Ponics_pomp_poliv				AT  %MB392	:	BOOL;	(*12484*)
	Ponics_time_elapsed_poliv			AT  %MB394	:	UINT;	(*12485*)
	Ponics_doliv_water_active			AT  %MB396	:	BOOL;	(*12486*)
	Ponics_doliv_AB_active			AT  %MB398	:	BOOL;	(*12487*)
 PONIC old1 *)


	Smoke_1floor					AT %MB400	:	BOOL;	(*12288+200=12488*)
	Smoke_2floor					AT %MB402	:	BOOL;	(*12489*)
	Smoke_sport					AT %MB404	:	BOOL;	(*12490*)
	Smoke_stair					AT %MB406	:	BOOL;	(*12491*)
	PIR_north_zapad				AT %MB408	:	BOOL;	(*12492*)
	PIR_north_vostok				AT %MB410	:	BOOL;	(*12493*)
	Gerkon_sklad				AT %MB412	:	BOOL;	(*12494*)
	Gerkon_door					AT %MB414	:	BOOL;	(*12495*)
	Light_reserv					AT %MB416	:	BOOL;	(*12496*)
	Light_reserv_manual			AT %MB418	:	INT;		(*12497*)
	Supply_akb					AT %MW420	:	REAL;	(*12498*)
	Security_delay				AT %MB424	:	INT;		(*12500*)
	Balkon_temp					AT %MW428 :	REAL; 	(*12502*)			(* PT1000 *)
	DC_Uv						AT %MW432 :	REAL; 	(*12504*)
	DC_Ia						AT %MW436 :	REAL; 	(*12506*)

	Teplica_tank_heat				AT %MB440	:	BOOL;	(*12508*)
	Teplica_set_temp_tank		AT %MB442	:	INT;		(*12509*)
	Teplica_set_finish_clear_vol	AT %MB444	:	INT:=10;	(*12510*)
	Teplica_set_finish_clear_time	AT %MB446	:	INT:=5;	(*12511*)
	Balkon_set_temp				AT  %MB448	:	UINT:=18;	(*12512*)
	Balkon_set_temp_day			AT  %MB450	:	UINT:=18;	(*12512*)
	Balkon_set_temp_night			AT  %MB452	:	UINT:=18;	(*12512*)

(* PONIC old2
	Ponics_pomp_doliv_water		AT  %MB450	:	BOOL;	(*12513*)
	Ponics_pomp_doliv_A			AT  %MB452	:	BOOL;	(*12514*)
	Ponics_pomp_doliv_B			AT  %MB454	:	BOOL;	(*12515*)
	Ponics_tank_water_level		AT  %MB456	:	BOOL;	(*12516*)
	Ponics_water_kf				AT  %MB458	:	UINT;	(*12517*)
	Ponics_A_kf					AT  %MB460	:	UINT;	(*12518*)
	Ponics_B_kf					AT  %MB462	:	UINT;	(*12519*)
	Ponics_status_PLC			AT  %MB464	:	UINT;	(*12520*)

	Ponics_set_doliv_A			AT  %MW468	:	REAL:=0.1;	(*12522*)
	Ponics_set_doliv_B			AT  %MW472	:	REAL:=0.1;	(*12524*)
	Ponics_set_doliv_water		AT  %MW476	:	REAL:=10;	(*12526*)
	Ponics_set_EC				AT  %MW480	:	REAL;	(*12528*)
	Ponics_EC					AT  %MW484	:	REAL;	(*12530*)
	Ponics_PH					AT  %MW488	:	REAL;	(*12532*)
	Ponics_tank_temp				AT  %MW492	:	REAL;	(*12534*)
	Ponics_tank_water_level_high	AT  %MB496	:	BOOL;	(*12536*)
 PONIC old2 *)

(*	Ponics_2						AT  %MW496	:	REAL;	(*12536*)
*)

	Poliv_zapad_minutes_est		AT %MB500	:	INT;		(*12288+250=12538*)
	Poliv_terrasa_minutes_est		AT %MB502	:	INT;		(*12539*)
	Poliv_south_minutes_est		AT %MB504	:	INT;		(*12540*)
	Poliv_north_minutes_est		AT %MB506	:	INT	;	(*12541 *)

	Kitchen_room_CO2			AT %MB508	:	INT;		(*12542 *)

	PLC_uptime					AT %MW512	:	DINT;	(*12544 *)

	RS485_1_cnt_success			AT %MW516	:	DINT;	(*12546 *)
	RS485_1_cnt_error			AT %MW520	:	DINT;	(*12548 *)
	RS485_2_cnt_success			AT %MW524	:	DINT;	(*12550 *)
	RS485_2_cnt_error			AT %MW528	:	DINT;	(*12552 *)
	RS485_3_cnt_success			AT %MW532	:	DINT;	(*12554 *)
	RS485_3_cnt_error			AT %MW536	:	DINT;	(*12556 *)
	Alarm_act					AT %MB540	:	INT;		(*12558 *)
	Alarm_button					AT %MB542	:	INT;		(*12559 *)
	Smoke_3floor					AT %MB544	:	BOOL;	(*12560*)
	Smoke_sklad					AT %MB546	:	BOOL;	(*12561*)
	Smoke_drovnik				AT %MB548	:	BOOL;	(*12562*)

	Teplica_temp_air				AT %MW552	:	REAL;	(*12564*)
	Teplica_temp_ground			AT %MW556	:	REAL;	 (*12566*)
	Teplica_light_lux				AT %MW560	:	REAL;	(*12568*)
	Teplica_temp_air_in			AT  %MW564:	REAL;       (*12570*)
	Teplica_temp_panel			AT %MW568	:	REAL;	(*12572*) (* Teplica_temp_panel*)
	Teplica_temp_LED			AT %MW572	:	REAL;	(*12574*)(* Teplica_temp_LED*)
	Teplica_t6					AT %MW576	:	REAL;	(*12576*)
	Teplica_t7					AT %MW580	:	REAL;	(*12578*)
	Teplica_max_EC				AT %MW584	:	REAL;	(*12580*)

	Teplica_impulse_water_cnt		AT %MW588	:	UDINT;		(*12582 16678*)
	Teplica_impulse_fertA_cnt		AT %MW592	:	UDINT;		(*12584 *)
	Teplica_impulse_fertB_cnt		AT %MW596	:	UDINT;		(*12586*)
	Teplica_fert_kf				AT %MB600	:	INT:=12;			(*12588*)

	Teplica_avg_lux				AT %MW604	:	REAL;		(*12590*)
	Teplica_fert_actA				AT %MW608	:	REAL;		(*12592*)
	Teplica_fert_actB				AT %MW612	:	REAL;		(*12594*)
(*	Teplica_DI8					AT %MB616	:	UDINT;	*)	(*12596*)

	Teplica_vent					AT %MB620	:	BOOL;		(*12598*)
	Teplica_heat					AT %MB622	:	BOOL;		(*12599*)
	Teplica_light					AT %MB624	:	BOOL;		(*12600*)
	Teplica_pomp_poliv			AT %MB626	:	BOOL;		(*12601*)
	Teplica_pomp_fertA			AT %MB628	:	BOOL;		(*12602*)
	Teplica_pomp_fertB			AT %MB630	:	BOOL;		(*12603*)
	Teplica_zone_poliv			AT %MB632	:	BOOL;		(*12604*)
	Teplica_DO8					AT %MB634	:	BOOL;		(*12605*)

	Teplica_temp_set_high		AT %MB636	:	INT:=21;		(*12606*)
	Teplica_temp_set_low			AT %MB638	:	INT:=18;		(*12607*)
	Teplica_light_set_low			AT %MW640	:	UINT:=10000;		(*12608*)
	Teplica_light_allow			AT %MB642	:	BOOL;	(*12609*)
	Teplica_poliv_active			AT %MB644	:	BOOL;	(*    BUTTON 12610*)

	Teplica_poliv_kf				AT %MB646	:	INT:=1030;	(*12611*)
	Teplica_fertA_kf				AT %MB648	:	INT:=10200;	(*12612*)
	Teplica_fertB_kf				AT %MB650	:	INT:=8700;	(*12613*)

	Teplica_set_poliv				AT %MW652	:	REAL:=200;	(*12614*)
	Teplica_set_fertA				AT %MW656	:	REAL:=1;	(*12616*)
	Teplica_set_fertB				AT %MW660	:	REAL:=1;	(*12618*)

	Teplica_time_elapsed_poliv	AT %MW664	:	UDINT;	(*12620*)
	Teplica_time_elapsed_fertA	AT %MW668	:	UDINT;	(*12622*)
	Teplica_time_elapsed_fertB	AT %MW672	:	UDINT;	(*12624*)

	Teplica_poliv_status_PLC		AT %MB676	:	INT;	(*12626*)
	Teplica_poliv_break			AT %MB678	:	BOOL;	(*12627*)

	Cnt_water_fertA				AT %MW680	:	UDINT;	(*12628		*)
	Cnt_water_fertB				AT %MW684	:	UDINT;	(*12630		*)


	Teplica_set_max_poliv_time	AT %MW688	:	UDINT:=60;	(*12632		*)
	Teplica_set_max_fertA_time	AT %MW692	:	UDINT:=10;	(*12634		*)
	Teplica_set_max_fertB_time	AT %MW696	:	UDINT:=10;	(*12636		*)
	Teplica_set_clear_time		AT %MW700	:	UDINT:=5;								(*12638		*)

	Balkon_light_lux				AT %MW704	:	UDINT;	(*12640		*)

	Balkon_light_rassada			AT %MB708	:	BOOL;		(*12642*)
	Balkon_light_rassada_allow	AT %MB710	:	BOOL;		(*12643*)
	Teplica_poliv_message_PLC	AT %MB712	:	INT:=0;		(*12644*)
	Teplica_power_light_lux		AT %MB714	:	INT:=20000;		(*12645*)
	Balkon_power_light_lux		AT %MB716	:	INT:=10000;		(*12646*)

	Teplica_temp_SHT30			AT %MW720	:	REAL;	(*12648*)
	Teplica_hum_SHT30			AT %MW724	:	REAL;	(*12650*)
	Teplica_temp_pipe_heat		AT %MW728	:	REAL;	(**) (*12652*)
	Teplica_sensor_soil_PH		AT %MW732	:	REAL;	(*12654*)
	Teplica_sensor_soil_EC		AT %MW736	:	REAL;	(*12656*)
	Teplica_sensor_soil_temp		AT %MW740	:	REAL;	(*12658*)
	Teplica_sensor_soil_hum		AT %MW744	:	REAL;	(*12660*)
	Teplica_sensor_soil_PH2		AT %MW748	:	REAL;	(*12662*)
	Teplica_temp_water_tank		AT %MW752	:	REAL;	(*12664*)
	Teplica_type_fert				AT %MB756	:	BOOL;	(*12666*)
	Teplica_type_poliv			AT %MB758	:	BOOL;	(*12667*)
	Teplica_tank_teplica_level		AT %MB760	:	BOOL;	(*12668*)
	Teplica_valve_water_in		AT %MB762	:	BOOL;	(*12669*) (*Teplica_valve_water_in*)
	Teplica_fert_pwm_levelA		AT %MB764	:	INT;		(*12670*)
	Teplica_fert_pwm_levelB		AT %MB766	:	INT;		(*12671*)
	Teplica_cnt_water_pipe		AT %MB768	:	INT;		(*12672*) (*Cnt_water_pipe*)
	Teplica_tank_level			AT %MB770	:	INT;		(*12673*) (*Teplica_tank_volume*)
	Teplica_tankA_level			AT %MB772	:	INT;		(*12674*)
	Teplica_tankB_level			AT %MB774	:	INT;		(*12675*)


(*          ***********PONICS*****************************                        *)

	Ponics_impulse_water_cnt			AT  %MW800	:	UDINT;	(* 400 +12288 = 12688*)
	Ponics_impulse_A_cnt				AT  %MW804	:	UDINT;	(*12690*)
	Ponics_impulse_B_cnt				AT  %MW808	:	UDINT;	(*12692*)
	Ponics_set_doliv_AB				AT  %MW812	:	REAL:=0.1;	(*12694*)
(*	Ponics_set_doliv_B				AT  %MW816	:	REAL:=0.1;*)	(*12696*)
	Ponics_set_doliv_water			AT  %MW820	:	REAL:=3;	(*12698*)
	Ponics_set_EC					AT  %MW824	:	REAL;	(*12700*)
	Ponics_EC						AT  %MW828	:	REAL;	(*12702*)
	Ponics_PH						AT  %MW832	:	REAL;	(*12704*)
	Ponics_tank_temp					AT  %MW836	:	REAL;	(*12706*)

	Ponics_set_max_poliv_time			AT  %MB840	:	UINT:=3000;	(*12708*)
	Ponics_set_max_doliv_water_time	AT  %MB842	:	UINT:=350;	(*12709*)
	Ponics_set_max_doliv_A_time		AT  %MB844	:	UINT:=20;	(*12710*)
	Ponics_set_max_doliv_B_time		AT  %MB846	:	UINT:=20;	(*12711*)
	Ponics_time_elapsed_poliv			AT  %MB848	:	UINT;	(*12712*)
	Ponics_water_kf					AT  %MB850	:	UINT:=11800;	(*12713*)
	Ponics_A_kf						AT  %MB852	:	UINT:=11700;	(*12714*)
	Ponics_B_kf						AT  %MB854	:	UINT:=12200;	(*12715*)
	Ponics_status_PLC				AT  %MB856	:	UINT;	(*12716*)

	Ponics_poliv_active				AT  %MB858	:	BOOL;	(*12717*)
	Ponics_poliv_break				AT  %MB860	:	BOOL;	(*12718*)
	Ponics_pomp_poliv				AT  %MB862	:	BOOL;	(*12719*)
	Ponics_doliv_water_active			AT  %MB864	:	BOOL;	(*12720*)
	Ponics_doliv_AB_active			AT  %MB866	:	BOOL;	(*12721*)
	Ponics_pomp_doliv_water			AT  %MB868	:	BOOL;	(*12722*)
	Ponics_pomp_doliv_A				AT  %MB870	:	BOOL;	(*12723*)
	Ponics_pomp_doliv_B				AT  %MB872	:	BOOL;	(*12724*)
	Ponics_tank_water_level			AT  %MB874	:	BOOL;	(*12725*)
	Ponics_tank_water_level_high		AT  %MB876	:	BOOL;	(*12288+438=12726*)

	Ponics_poliv_start					AT  %MW880	:	UDINT:=	25200000;	(*12728*) (*12288+440=12728*)
	Ponics_poliv_end					AT  %MW884	:	UDINT:=	25200000;	(*12730*)
	Ponics_doliv_AB_start				AT  %MW888	:	UDINT:=	25200000;	(*12732*)
	Ponics_doliv_AB_end				AT  %MW892	:	UDINT:=	25200000;	(*12734*)
	Ponics_doliv_water_start			AT  %MW896	:	UDINT:=	25200000;	(*12736*)
	Ponics_doliv_water_end			AT  %MW900	:	UDINT:=	25200000;	(*12738*)
	Ponics_light_morning_start			AT  %MW904	:	UDINT:=	25200000;	(*12740*)
	Ponics_light_morning_end			AT  %MW908	:	UDINT:=	25200000;	(*12288+454=12742*)
	Ponics_start_mintutes_poliv			AT  %MB912	:	UINT:=0;	(*12744*)
	Ponics_start_minutes_doliv_AB		AT  %MB914	:	UINT:=30;	(*12745*)
	Ponics_start_minutes_doliv_water	AT  %MB916	:	UINT:=20;	(*12746*)

	Ponics_time_elapsed_doliv_A		AT  %MW920	:	UDINT:=0;	 (*12288+460=12748*)
	Ponics_time_elapsed_doliv_B		AT  %MW924	:	UDINT:=0;	 (*12288+462=12750*)
	Ponics_time_elapsed_doliv_water	AT  %MW928	:	UDINT:=0;	(*12752*)
	Balkon_hum						AT  %MW932	:	REAL;	(*12754*)

	Sensor_EC2						AT  %MW936	:	REAL;	(*12756*)
	Sensor_house_water_imp			AT  %MW940	:	UDINT;  (*12758*)
	Modbus_4errors					AT  %MW944	:	UDINT; (*12760*)
	Modbus_qual_errors				AT  %MW948	:	UINT; (*12762*)
	Balkon_CO2						AT  %MW950	:	UINT; (*12763*)
	Teplica_CO2						AT  %MW952	:	UINT; (*12764*)
	Teplica_pwm_avg_A				AT  %MW956	:	REAL; (*12766*)
	Teplica_pwm_avg_B				AT  %MW960	:	REAL; (*12768*)
	Battery_low						AT  %MB964	:	BOOL; (*12770*)

(*          ***********PARNIK*****************************                        *)
	Parnik_air_temp					AT %MW968	:	REAL;	(*12772*)
	Parnik_ground_temp				AT %MW972	:	REAL;	(*12774*)
	Parnik_sht_air_hum				AT %MW976	:	REAL;	(*12776*)
	Parnik_sht_air_temp				AT %MW980	:	REAL;	(*12778*)
	Parnik_manual_level_window	AT %MW984	:	INT;		(*12780*)
	Parnik_current_level_window	AT %MW986	:	INT;		(*12781*)
	Parnik_temp_step1_window		AT %MW988	:	INT;		(*12782*)
	Parnik_temp_step2_window		AT %MW990	:	INT;		(*12783*)
	Parnik_set_auto_window		AT %MW992	:	BOOL;	(*12784*)
	Parnik_set_temp_street_min	AT %MW994	:	INT;		(*12785*)
	Parnik_pipe_temp				AT %MW1000	:	REAL;	(*12788*)




(*	Teplica_impulse_water_cnt			AT %MW368	:	UDINT;	(*12472*)
	Teplica_impulse_fertA_cnt			AT %MW372	:	UDINT;	(*12474*)
	Teplica_impulse_fertB_cnt			AT %MW376	:	UDINT;	(*12476*)
*)
(*
	Teplica_vent						AT %MB380	:	BOOL;		(*12478*)
	Teplica_heat						AT %MB382	:	BOOL;		(*12479*)
	Teplica_light						AT %MB384	:	BOOL;		(*12480*)
	Teplica_pomp_poliv				AT %MB386	:	BOOL;		(*12481*)
	Teplica_pomp_fertA				AT %MB388	:	BOOL;		(*12482*)
	Teplica_pomp_fertB				AT %MB390	:	BOOL;		(*12483*)
*)
















(*
	M1T1					AT %MB600	:	REAL;
	M1T2					AT %MB604	:	REAL;
	M2T1					AT %MB608	:	REAL;
	M2T2					AT %MB612	:	REAL;
	M3T1					AT %MB616	:	REAL;
	M3T2					AT %MB620	:	REAL;
	M4T1					AT %MB624	:	REAL;
	M4T2					AT %MB628	:	REAL;
	M5T1					AT %MB632	:	REAL;
	M5T2					AT %MB636	:	REAL;
	M6T1					AT %MB640	:	REAL;
	M6T2					AT %MB644	:	REAL;
	M7T1					AT %MB648	:	REAL;
	M7T2					AT %MB652	:	REAL;
	M8T1					AT %MB656	:	REAL;
	M8T2					AT %MB660	:	REAL;
	M9T1					AT %MB664	:	REAL;
	M9T2					AT %MB668	:	REAL;
	M10T1					AT %MB672	:	REAL;
	M10T2					AT %MB676	:	REAL;
	M11T1					AT %MB680	:	REAL;
	M11T2					AT %MB684	:	REAL;
	M12T1					AT %MB688	:	REAL;
	M12T2					AT %MB692	:	REAL;
*)

END_STRUCT
END_TYPE

(* Data type *)
TYPE ST_MqttReceivedPublishTelegram :
STRUCT
	sTopic		: STRING[255];
	sValue		: STRING[255];
	bHasData	: BOOL;
END_STRUCT
END_TYPE

(* Data type *)
TYPE ST_MqttSettings :
STRUCT
	(* informations *)
	sMqttClientId	: STRING[23];
	sMqttUserId	: STRING[25];
	sMqttPassword	: STRING[25];
	sMqttBrokerIP	: STRING[15];
	nMqttBrokerPort	: UDINT := 1883;

	(* state *)
	bSocketConnection	: BOOL := FALSE;
	bConnected			: BOOL := FALSE;
	bConnectPackageSent	: BOOL := FALSE;
	bDisconnect			: BOOL := FALSE;
	bError				: BOOL := FALSE;
	bValidConnection	: BOOL := FALSE;
	bActive				: BOOL := FALSE;
	wPackageIdentifier	: WORD := 1;
	hSocket				: T_HSOCKET;
	tonSendPingReq		: TON;

	(* send *)
	stMqttSendTelegram			: ST_MqttTelegram;
	stMqttLastSendTelegram		: ST_MqttTelegram;

	(* receive *)
	stMqttReceivedTelegram			: ST_MqttTelegram;
	stMqttLastReceivedTelegram		: ST_MqttTelegram;
	stMqttReceivedPublishTelegram	: ST_MqttReceivedPublishTelegram;

	(* settings internal *)
	iTelegramSize	: INT := 544;
	usKeepAliveTime	: USINT := 60; (* seconds *)

END_STRUCT
END_TYPE

(* Data type *)
TYPE ST_MqttTelegram :
STRUCT
	arMqttData 	: ARRAY[0..544] OF BYTE;
	nDataLength	: UDINT := 0;
END_STRUCT
END_TYPE

(* Data type *)
TYPE stIobroker :
STRUCT

	Control_hum					:	REAL;
	Control_temp					:	REAL;
	Control_hum2					:	REAL;
	Control_temp2				:	REAL;

END_STRUCT
END_TYPE

(* Data type *)
TYPE stMB :
STRUCT

	M1T1							AT %MW0	:REAL;  	(* modbus address 12288 *)
	M1T2							AT %MW4	:REAL;	(* 12290 *)
	M2T1							AT %MW8	:REAL;	(* 12292 *)
	M2T2							AT %MW12	:REAL;	 (* 12294 *)
	M3T1							AT %MW16	:REAL;	 (* 12296 *)
	M3T2							AT %MW20	:REAL;	 (* 12298 *)
	M4T1							AT %MW24	:REAL;	 (* 12300 *)
	M4T2							AT %MW28	:REAL;	 (* 12302 *)
	M5T1							AT %MW32	:REAL;	 (* 12304 *)
	M5T2							AT %MW36	:REAL;	 (* 12306 *)
	M6T1							AT %MW40	:REAL;	 (* 12308 *)
	M6T2							AT %MW44	:REAL;	(* 12310 *)
	M7T1							AT %MW48	:REAL;	 (* 12312 *)
	M7T2							AT %MW52	:REAL;	 (* 12314 *)
	M8T1							AT %MW56	:REAL;	 (* 12316 *)
	M8T2							AT %MW60	:REAL;	(* 12318 *)
	M9T1							AT %MW64	:REAL;	(* 12320 *)
	M9T2							AT %MW68	:REAL;	(* 12322 *)
	M10T1							AT %MW72	:REAL;	(* 12324 *)
	M10T2							AT %MW76	:REAL;	(* 12326 *)
	M11T1							AT %MW80	:REAL;	(* 12328 *)
	M11T2							AT %MW84	:REAL;	(* 12330 *)
	M12T1							AT %MW88	:REAL;	(* 12332 *)
	M12T2							AT %MW92	:REAL;	(* 12334 *)

END_STRUCT
END_TYPE

(* Data type *)
TYPE stMercury :
STRUCT

	M1T1					:	REAL;
	M1T2					:	REAL;
	M2T1					:	REAL;
	M2T2					:	REAL;
	M3T1					:	REAL;
	M3T2					:	REAL;
	M4T1					:	REAL;
	M4T2					:	REAL;
	M5T1					:	REAL;
	M5T2					:	REAL;
	M6T1					:	REAL;
	M6T2					:	REAL;
	M7T1					:	REAL;
	M7T2					:	REAL;
	M8T1					:	REAL;
	M8T2					:	REAL;
	M9T1					:	REAL;
	M9T2					:	REAL;
	M10T1					:	REAL;
	M10T2					:	REAL;
	M11T1					:	REAL;
	M11T2					:	REAL;
	M12T1					:	REAL;
	M12T2					:	REAL;

END_STRUCT
END_TYPE

(* POU MAIN, ST *)
PROGRAM MAIN
VAR

(*	ToFromNovRam2			AT %Q*:DataToFromNovram2; *)
(*	ToFromNovRam			AT %QB200:DataToFromNovram; *)
(*	ToFromNovRam			AT %Q*:DataToFromNovram; *)
	INITVAR					: BOOL:=FALSE;




END_VAR
(*
IF (INITVAR=FALSE) THEN

	(* START RESTORE VARS FROM MEMORY AFTER REBOOT/RESET/LOST POWER *)

	Modbus.Target_CO2				:=	ToFromNovRam.Target_CO2_mem;
	Modbus.First_floor_temp_target		:=	ToFromNovRam.First_floor_temp_target_mem;
	Modbus.Second_floor_temp_target	:=	ToFromNovRam.Second_floor_temp_target_mem;
	Modbus.Sport_temp_target			:=	ToFromNovRam.Sport_temp_target_mem;
	Modbus.Sauna_temp_target		:=	ToFromNovRam.Sauna_temp_target_mem;

	Modbus.Underfloor_temp_target		:=	ToFromNovRam.Underfloor_temp_target_mem;
	Modbus.Underfloor_humidity_target	:=	ToFromNovRam.Underfloor_humidity_target_mem;

	Modbus.Vent						:=	ToFromNovRam.Vent_mem;
	Modbus.Vent_heat				:=	ToFromNovRam.Vent_heat_mem;
	Modbus.Vent_heat_level			:=	ToFromNovRam.Vent_heat_level_mem;

	Modbus.Pomp_house				:=	ToFromNovRam.Pomp_house_mem;
	Modbus.Pomp_garden				:=	ToFromNovRam.Pomp_garden_mem;
	Modbus.Light_garden				:=	ToFromNovRam.Light_garden_mem;

	Modbus.Poliv_zapad_minutes		:=	ToFromNovRam.Poliv_zapad_minutes;
	Modbus.Poliv_terrasa_minutes		:=	ToFromNovRam.Poliv_terrasa_minutes;
	Modbus.Poliv_south_minutes		:=	ToFromNovRam.Poliv_south_minutes;
	Modbus.Poliv_north_minutes		:=	ToFromNovRam.Poliv_north_minutes;

	Modbus.Teplica_temp_set_high		:=	ToFromNovRam.Teplica_temp_set_high;
	Modbus.Teplica_temp_set_low		:=	ToFromNovRam.Teplica_temp_set_low;
	Modbus.Teplica_light_set_low		:=	ToFromNovRam.Teplica_light_set_low;
	Modbus.Teplica_light_allow			:=	ToFromNovRam.Teplica_light_allow;
	Modbus.Teplica_poliv_kf			:=	ToFromNovRam.Teplica_poliv_kf;
	Modbus.Teplica_fertA_kf			:=	ToFromNovRam.Teplica_fertA_kf;
	Modbus.Teplica_fertB_kf			:=	ToFromNovRam.Teplica_fertB_kf;
	Modbus.Teplica_set_poliv			:=	ToFromNovRam.Teplica_set_poliv;
	Modbus.Teplica_set_fertA			:=	ToFromNovRam.Teplica_set_fertA;
	Modbus.Teplica_set_fertB			:=	ToFromNovRam.Teplica_set_fertB;
	Modbus.Teplica_set_max_poliv_time	:=	ToFromNovRam.Teplica_set_max_poliv_time;
	Modbus.Teplica_set_max_fertA_time	:=	ToFromNovRam.Teplica_set_max_fertA_time;
	Modbus.Teplica_set_max_fertB_time	:=	ToFromNovRam.Teplica_set_max_fertB_time;
	Modbus.Teplica_set_max_fertB_time	:=	ToFromNovRam.Teplica_set_clear_time;
	Modbus.Teplica_set_temp_pomp_cold	:=	ToFromNovRam.Teplica_set_temp_pomp_cold;
	Modbus.Teplica_set_temp_window_open	:=	ToFromNovRam.Teplica_set_temp_window_open;
	Modbus.Teplica_set_poliv_before_fert	:=	ToFromNovRam.Teplica_set_poliv_before_fert;

	Modbus.Teplica_set_temp_tank			:=	ToFromNovRam.Teplica_set_temp_tank;
	Modbus.Teplica_fert_kf				:=	ToFromNovRam.Teplica_fert_kf;
	Modbus.Teplica_zone_poliv			:=	ToFromNovRam.Teplica_zone_poliv;
	Modbus.Teplica_type_fert				:=	ToFromNovRam.Teplica_type_fert;
	Modbus.Teplica_type_poliv				:=	ToFromNovRam.Teplica_type_poliv;
	Modbus.Teplica_set_clear_time			:=	ToFromNovRam.Teplica_set_clear_time;
	Modbus.Teplica_set_finish_clear_time	:=	ToFromNovRam.Teplica_set_finish_clear_time;
	Modbus.Teplica_set_finish_clear_vol		:=	ToFromNovRam.Teplica_set_finish_clear_vol;

	Modbus.Ponics_start_mintutes_poliv			:=	ToFromNovRam.Ponics_start_mintutes_poliv;
	Modbus.Ponics_start_minutes_doliv_AB		:=	ToFromNovRam.Ponics_start_minutes_doliv_AB;
	Modbus.Ponics_start_minutes_doliv_water	:=	ToFromNovRam.Ponics_start_minutes_doliv_water;
	Modbus.Ponics_set_doliv_A				:=	ToFromNovRam.Ponics_set_doliv_A;
	Modbus.Ponics_set_doliv_water				:=	ToFromNovRam.Ponics_set_doliv_water;
	Modbus.Ponics_set_max_poliv_time			:=	ToFromNovRam.Ponics_set_max_poliv_time;
	Modbus.Ponics_set_max_doliv_A_time		:=	ToFromNovRam.Ponics_set_max_doliv_A_time;
	Modbus.Ponics_set_max_doliv_water_time	:=	ToFromNovRam.Ponics_set_max_doliv_water_time;
	Modbus.Balkon_set_temp					:=	ToFromNovRam.Balkon_set_temp;
	Modbus.Ponics_A_kf						:=	ToFromNovRam.Ponics_A_kf;
	Modbus.Ponics_B_kf						:=	ToFromNovRam.Ponics_B_kf;
	Modbus.Ponics_water_kf					:=	ToFromNovRam.Ponics_water_kf;


	(* END RESTORE VARS FROM MEMORY AFTER REBOOT/RESET/LOST POWER *)

	INITVAR:=TRUE;
ELSE
	(*START SAVE VARS to PERSISTENT MEMORY*)
	ToFromNovRam.Target_CO2_mem					:=	Modbus.Target_CO2;
	ToFromNovRam.First_floor_temp_target_mem		:=	Modbus.First_floor_temp_target;
	ToFromNovRam.Second_floor_temp_target_mem		:=	Modbus.Second_floor_temp_target;
	ToFromNovRam.Sport_temp_target_mem			:=	Modbus.Sport_temp_target;
	ToFromNovRam.Sauna_temp_target_mem			:=	Modbus.Sauna_temp_target;

	ToFromNovRam.Underfloor_temp_target_mem		:=	Modbus.Underfloor_temp_target;
	ToFromNovRam.Underfloor_humidity_target_mem	:=	Modbus.Underfloor_humidity_target;

	ToFromNovRam.Vent_mem						:=	Modbus.Vent;
	ToFromNovRam.Vent_heat_mem					:=	Modbus.Vent_heat;
	ToFromNovRam.Vent_heat_level_mem				:=	Modbus.Vent_heat_level;

	ToFromNovRam.Pomp_house_mem				:=	Modbus.Pomp_house;
	ToFromNovRam.Pomp_garden_mem				:=	Modbus.Pomp_garden;
	ToFromNovRam.Light_garden_mem				:=	Modbus.Light_garden;


	ToFromNovRam.Poliv_zapad_minutes			:=	Modbus.Poliv_zapad_minutes;
	ToFromNovRam.Poliv_terrasa_minutes			:=	Modbus.Poliv_terrasa_minutes;
	ToFromNovRam.Poliv_south_minutes			:=	Modbus.Poliv_south_minutes;
	ToFromNovRam.Poliv_north_minutes			:=	Modbus.Poliv_north_minutes;


	ToFromNovRam.Teplica_temp_set_high		:=	Modbus.Teplica_temp_set_high;
	ToFromNovRam.Teplica_temp_set_low			:=	Modbus.Teplica_temp_set_low;
	ToFromNovRam.Teplica_light_set_low			:=	Modbus.Teplica_light_set_low;
	ToFromNovRam.Teplica_light_allow			:=	Modbus.Teplica_light_allow;
	ToFromNovRam.Teplica_poliv_kf				:= 	Modbus.Teplica_poliv_kf;
	ToFromNovRam.Teplica_fertA_kf				:= 	Modbus.Teplica_fertA_kf;
	ToFromNovRam.Teplica_fertB_kf				:=	Modbus.Teplica_fertB_kf;
	ToFromNovRam.Teplica_set_poliv				:=	Modbus.Teplica_set_poliv;
	ToFromNovRam.Teplica_set_fertA				:=	Modbus.Teplica_set_fertA;
	ToFromNovRam.Teplica_set_fertB				:=	Modbus.Teplica_set_fertB;
	ToFromNovRam.Teplica_set_max_poliv_time	:=	Modbus.Teplica_set_max_poliv_time;
	ToFromNovRam.Teplica_set_max_fertA_time	:=	Modbus.Teplica_set_max_fertA_time;
	ToFromNovRam.Teplica_set_max_fertB_time	:=	Modbus.Teplica_set_max_fertB_time;
	ToFromNovRam.Teplica_set_clear_time		:=	Modbus.Teplica_set_max_fertB_time;
	ToFromNovRam.Teplica_set_temp_pomp_cold	:=	Modbus.Teplica_set_temp_pomp_cold;
	ToFromNovRam.Teplica_set_temp_window_open	:=	Modbus.Teplica_set_temp_window_open;
	ToFromNovRam.Teplica_set_poliv_before_fert	:=	Modbus.Teplica_set_poliv_before_fert;

	ToFromNovRam.Teplica_set_temp_tank		:=	Modbus.Teplica_set_temp_tank			;
	ToFromNovRam.Teplica_fert_kf				:=	Modbus.Teplica_fert_kf				;
	ToFromNovRam.Teplica_zone_poliv			:=	Modbus.Teplica_zone_poliv			;
	ToFromNovRam.Teplica_type_fert			:=	Modbus.Teplica_type_fert				;
	ToFromNovRam.Teplica_type_poliv			:=	Modbus.Teplica_type_poliv				;
	ToFromNovRam.Teplica_set_clear_time		:=	Modbus.Teplica_set_clear_time			;
	ToFromNovRam.Teplica_set_finish_clear_time	:=	Modbus.Teplica_set_finish_clear_time;
	ToFromNovRam.Teplica_set_finish_clear_vol		:=	Modbus.Teplica_set_finish_clear_vol	;

	ToFromNovRam.Ponics_start_mintutes_poliv			:=	Modbus.Ponics_start_mintutes_poliv;
	ToFromNovRam.Ponics_start_minutes_doliv_AB		:=	Modbus.Ponics_start_minutes_doliv_AB;
	ToFromNovRam.Ponics_start_minutes_doliv_water	:=	Modbus.Ponics_start_minutes_doliv_water;
	ToFromNovRam.Ponics_set_doliv_A				:=	Modbus.Ponics_set_doliv_A;
	ToFromNovRam.Ponics_set_doliv_water				:=	Modbus.Ponics_set_doliv_water;
	ToFromNovRam.Ponics_set_max_poliv_time			:=	Modbus.Ponics_set_max_poliv_time;
	ToFromNovRam.Ponics_set_max_doliv_A_time		:=	Modbus.Ponics_set_max_doliv_A_time;
	ToFromNovRam.Ponics_set_max_doliv_water_time	:=	Modbus.Ponics_set_max_doliv_water_time;
	ToFromNovRam.Balkon_set_temp					:=	Modbus.Balkon_set_temp;
	ToFromNovRam.Ponics_A_kf						:=	Modbus.Ponics_A_kf;
	ToFromNovRam.Ponics_B_kf						:=	Modbus.Ponics_B_kf;
	ToFromNovRam.Ponics_water_kf					:=	Modbus.Ponics_water_kf;


*)


	(*END SAVE VARS to PERSISTENT MEMORY*)
	fast;


(*
	Sensors;						(* Аналогвые датчики на шине KL *)
	Security_new;						(* Мониторинг датчиков охраны *)
	RS485read;					(* Опрос устройств на шине RS485 *)
	RS485read_2;					(* Опрос устройств на шине RS485 *)
	RS485read_3;					(* Опрос устройств на шине RS485 *)

	VentControl;					(* Глобальный контроль вентустановки*)
	VentPower;					(* Авторегулировка мощности вентустановки по датчикам CO2*)
	Poliv;						(* Таймеры зонального полива *)


	Power_act;					(*Контроль резервного освещения*)
	Alarm;


(* Прямое присовение виртуальных переменных к переменным, жестко привязаным к физ. портам. Частота обновления= циклу ПЛК (50 мсек) : *)
	HW_pomp_house				:=	Modbus.Pomp_house;
	Modbus.Sensor_supply		:=	HW_sensor_supply;
	HW_kalitka					:=	Modbus.Kalitka;
	iobroker.button_light_garden	:=	HW_button_light_garden;
	HW_light_garden				:=	Modbus.Light_garden;
	iobroker.Light_garden			:=	Modbus.Light_garden;
	Modbus.Valve_status			:=	BOOL_TO_INT(HW_vent_relay_pressure);
	Modbus.Balkon_light_rassada	:=	HW_light_rassada;

	Buttons;						(*Обработка нажатия кнопок *)
	tmCheck();
	tmCheckE();
	Timer_day();
	Timer_CO2();
	tmcheckM();

	Modbus.PLC_uptime			:=	SystemTaskInfoArr[1].cycleCount;
	HW_teplica_pomp_fert_level	:=	Modbus.Teplica_pomp_fert_level;
	HW_teplica_pomp_poliv	:=	Modbus.Teplica_pomp_poliv;
	IF (Modbus.Teplica_pomp_fertA = TRUE OR Modbus.Teplica_pomp_fertB = TRUE) THEN
		HW_teplica_pomp_fertA	:=	TRUE;
	ELSE
				HW_teplica_pomp_fertA	:=	FALSE;
	END_IF
	HW_teplica_zone_poliv	:=	Modbus.Teplica_zone_poliv;
*)

(*
END_IF
*)
END_PROGRAM

(* POU Intern/fast, ST *)
PROGRAM fast
VAR
END_VAR
Trigger_water_impulse_ponics(CLK:=HW_impulse_water_ponics);
Trigger_A_impulse_Ponics(CLK:=HW_impulse_tankA_Ponics);
Trigger_B_impulse_Ponics(CLK:=HW_impulse_tankB_Ponics);

Trigger_water_impulse_teplica(CLK:=HW_impulse_water_teplica);
Trigger_fertA_impulse_teplica(CLK:=HW_impulse_fertA_teplica);
Trigger_fertB_impulse_teplica(CLK:=HW_impulse_fertB_teplica);



IF Trigger_water_impulse_Ponics.Q THEN
	Modbus.Ponics_impulse_water_cnt	:= 	Modbus.Ponics_impulse_water_cnt+1;
END_IF

IF Trigger_A_impulse_Ponics.Q THEN
	Modbus.Ponics_impulse_A_cnt	:= 	Modbus.Ponics_impulse_A_cnt+1;
END_IF
IF Trigger_B_impulse_Ponics.Q THEN
	Modbus.Ponics_impulse_B_cnt	:= 	Modbus.Ponics_impulse_B_cnt+1;
END_IF



IF Trigger_water_impulse_teplica.Q THEN
	Modbus.Teplica_impulse_water_cnt	:= 	Modbus.Teplica_impulse_water_cnt+1;
END_IF


IF Trigger_fertA_impulse_teplica.Q THEN
	Modbus.Teplica_impulse_fertA_cnt	:= 	Modbus.Teplica_impulse_fertA_cnt+1;
END_IF
IF Trigger_fertB_impulse_teplica.Q THEN
	Modbus.Teplica_impulse_fertB_cnt	:= 	Modbus.Teplica_impulse_fertB_cnt+1;
END_IF
END_PROGRAM

(* POU MAIN2, ST *)
PROGRAM MAIN2
VAR
	i: INT;
	ToFromNovRam			AT %Q*:DataToFromNovram;
	INITVAR					: BOOL:=FALSE;

END_VAR
IF (INITVAR=FALSE) THEN

	(* START RESTORE VARS FROM MEMORY AFTER REBOOT/RESET/LOST POWER *)

	Modbus.Target_CO2				:=	ToFromNovRam.Target_CO2_mem;
	Modbus.First_floor_temp_target		:=	ToFromNovRam.First_floor_temp_target_mem;
	Modbus.Second_floor_temp_target	:=	ToFromNovRam.Second_floor_temp_target_mem;
	Modbus.Sport_temp_target			:=	ToFromNovRam.Sport_temp_target_mem;
	Modbus.Sauna_temp_target		:=	ToFromNovRam.Sauna_temp_target_mem;

	Modbus.Underfloor_temp_target		:=	ToFromNovRam.Underfloor_temp_target_mem;
	Modbus.Underfloor_humidity_target	:=	ToFromNovRam.Underfloor_humidity_target_mem;

	Modbus.Vent						:=	ToFromNovRam.Vent_mem;
	Modbus.Vent_heat				:=	ToFromNovRam.Vent_heat_mem;
	Modbus.Vent_heat_level			:=	ToFromNovRam.Vent_heat_level_mem;

	Modbus.Pomp_house				:=	ToFromNovRam.Pomp_house_mem;
	Modbus.Pomp_garden				:=	ToFromNovRam.Pomp_garden_mem;
	Modbus.Light_garden				:=	ToFromNovRam.Light_garden_mem;

	Modbus.Poliv_zapad_minutes		:=	ToFromNovRam.Poliv_zapad_minutes;
	Modbus.Poliv_terrasa_minutes		:=	ToFromNovRam.Poliv_terrasa_minutes;
	Modbus.Poliv_south_minutes		:=	ToFromNovRam.Poliv_south_minutes;
	Modbus.Poliv_north_minutes		:=	ToFromNovRam.Poliv_north_minutes;

	Modbus.Teplica_temp_set_high		:=	ToFromNovRam.Teplica_temp_set_high;
	Modbus.Teplica_temp_set_low		:=	ToFromNovRam.Teplica_temp_set_low;
	Modbus.Teplica_light_set_low		:=	ToFromNovRam.Teplica_light_set_low;
	Modbus.Teplica_light_allow			:=	ToFromNovRam.Teplica_light_allow;
	Modbus.Teplica_poliv_kf			:=	ToFromNovRam.Teplica_poliv_kf;
	Modbus.Teplica_fertA_kf			:=	ToFromNovRam.Teplica_fertA_kf;
	Modbus.Teplica_fertB_kf			:=	ToFromNovRam.Teplica_fertB_kf;
	Modbus.Teplica_set_poliv			:=	ToFromNovRam.Teplica_set_poliv;
	Modbus.Teplica_set_fertA			:=	ToFromNovRam.Teplica_set_fertA;
	Modbus.Teplica_set_fertB			:=	ToFromNovRam.Teplica_set_fertB;
	Modbus.Teplica_set_max_poliv_time	:=	ToFromNovRam.Teplica_set_max_poliv_time;
	Modbus.Teplica_set_max_fertA_time	:=	ToFromNovRam.Teplica_set_max_fertA_time;
	Modbus.Teplica_set_max_fertB_time	:=	ToFromNovRam.Teplica_set_max_fertB_time;
	Modbus.Teplica_set_max_fertB_time	:=	ToFromNovRam.Teplica_set_clear_time;
	Modbus.Teplica_set_temp_pomp_cold	:=	ToFromNovRam.Teplica_set_temp_pomp_cold;
	Modbus.Teplica_set_temp_window_open	:=	ToFromNovRam.Teplica_set_temp_window_open;
	Modbus.Teplica_set_poliv_before_fert	:=	ToFromNovRam.Teplica_set_poliv_before_fert;

	Modbus.Teplica_set_temp_tank			:=	ToFromNovRam.Teplica_set_temp_tank;
	Modbus.Teplica_fert_kf				:=	ToFromNovRam.Teplica_fert_kf;
	Modbus.Teplica_zone_poliv			:=	ToFromNovRam.Teplica_zone_poliv;
	Modbus.Teplica_type_fert				:=	ToFromNovRam.Teplica_type_fert;
	Modbus.Teplica_type_poliv				:=	ToFromNovRam.Teplica_type_poliv;
	Modbus.Teplica_set_clear_time			:=	ToFromNovRam.Teplica_set_clear_time;
	Modbus.Teplica_set_finish_clear_time	:=	ToFromNovRam.Teplica_set_finish_clear_time;
	Modbus.Teplica_set_finish_clear_vol		:=	ToFromNovRam.Teplica_set_finish_clear_vol;

	Modbus.Ponics_start_mintutes_poliv			:=	ToFromNovRam.Ponics_start_mintutes_poliv;
	Modbus.Ponics_start_minutes_doliv_AB		:=	ToFromNovRam.Ponics_start_minutes_doliv_AB;
	Modbus.Ponics_start_minutes_doliv_water	:=	ToFromNovRam.Ponics_start_minutes_doliv_water;
	Modbus.Ponics_set_doliv_AB				:=	ToFromNovRam.Ponics_set_doliv_AB;
	Modbus.Ponics_set_doliv_water				:=	ToFromNovRam.Ponics_set_doliv_water;
	Modbus.Ponics_set_max_poliv_time			:=	ToFromNovRam.Ponics_set_max_poliv_time;
	Modbus.Ponics_set_max_doliv_A_time		:=	ToFromNovRam.Ponics_set_max_doliv_A_time;
	Modbus.Ponics_set_max_doliv_water_time	:=	ToFromNovRam.Ponics_set_max_doliv_water_time;
	Modbus.Ponics_set_EC					:=	ToFromNovRam.Ponics_set_EC;
	Modbus.Balkon_set_temp					:=	ToFromNovRam.Balkon_set_temp;
	Modbus.Ponics_A_kf						:=	ToFromNovRam.Ponics_A_kf;
	Modbus.Ponics_B_kf						:=	ToFromNovRam.Ponics_B_kf;
	Modbus.Ponics_water_kf					:=	ToFromNovRam.Ponics_water_kf;
	Modbus.Sensor_house_water_imp			:=	ToFromNovRam.Sensor_house_water_imp;

	Modbus.Parnik_temp_step1_window			:=	ToFromNovRam.Parnik_temp_step1_window;
	Modbus.Parnik_temp_step2_window			:=	ToFromNovRam.Parnik_temp_step2_window;
	Modbus.Parnik_set_auto_window			:=	ToFromNovRam.Parnik_set_auto_window;
	Modbus.Parnik_current_level_window		:=	ToFromNovRam.Parnik_current_level_window;
	Modbus.Parnik_manual_level_window		:=	ToFromNovRam.Parnik_manual_level_window;


	(* END RESTORE VARS FROM MEMORY AFTER REBOOT/RESET/LOST POWER *)
(*
	pwm_ctrl_1	:= 2;
	fert_pwm_levelA	:= 491; *)

	INITVAR:=TRUE;
ELSE
	(*START SAVE VARS to PERSISTENT MEMORY*)
	ToFromNovRam.Target_CO2_mem					:=	Modbus.Target_CO2;
	ToFromNovRam.First_floor_temp_target_mem		:=	Modbus.First_floor_temp_target;
	ToFromNovRam.Second_floor_temp_target_mem		:=	Modbus.Second_floor_temp_target;
	ToFromNovRam.Sport_temp_target_mem			:=	Modbus.Sport_temp_target;
	ToFromNovRam.Sauna_temp_target_mem			:=	Modbus.Sauna_temp_target;

	ToFromNovRam.Underfloor_temp_target_mem		:=	Modbus.Underfloor_temp_target;
	ToFromNovRam.Underfloor_humidity_target_mem	:=	Modbus.Underfloor_humidity_target;

	ToFromNovRam.Vent_mem						:=	Modbus.Vent;
	ToFromNovRam.Vent_heat_mem					:=	Modbus.Vent_heat;
	ToFromNovRam.Vent_heat_level_mem				:=	Modbus.Vent_heat_level;

	ToFromNovRam.Pomp_house_mem				:=	Modbus.Pomp_house;
	ToFromNovRam.Pomp_garden_mem				:=	Modbus.Pomp_garden;
	ToFromNovRam.Light_garden_mem				:=	Modbus.Light_garden;


	ToFromNovRam.Poliv_zapad_minutes			:=	Modbus.Poliv_zapad_minutes;
	ToFromNovRam.Poliv_terrasa_minutes			:=	Modbus.Poliv_terrasa_minutes;
	ToFromNovRam.Poliv_south_minutes			:=	Modbus.Poliv_south_minutes;
	ToFromNovRam.Poliv_north_minutes			:=	Modbus.Poliv_north_minutes;


	ToFromNovRam.Teplica_temp_set_high		:=	Modbus.Teplica_temp_set_high;
	ToFromNovRam.Teplica_temp_set_low			:=	Modbus.Teplica_temp_set_low;
	ToFromNovRam.Teplica_light_set_low			:=	Modbus.Teplica_light_set_low;
	ToFromNovRam.Teplica_light_allow			:=	Modbus.Teplica_light_allow;
	ToFromNovRam.Teplica_poliv_kf				:= 	Modbus.Teplica_poliv_kf;
	ToFromNovRam.Teplica_fertA_kf				:= 	Modbus.Teplica_fertA_kf;
	ToFromNovRam.Teplica_fertB_kf				:=	Modbus.Teplica_fertB_kf;
	ToFromNovRam.Teplica_set_poliv				:=	Modbus.Teplica_set_poliv;
	ToFromNovRam.Teplica_set_fertA				:=	Modbus.Teplica_set_fertA;
	ToFromNovRam.Teplica_set_fertB				:=	Modbus.Teplica_set_fertB;
	ToFromNovRam.Teplica_set_max_poliv_time	:=	Modbus.Teplica_set_max_poliv_time;
	ToFromNovRam.Teplica_set_max_fertA_time	:=	Modbus.Teplica_set_max_fertA_time;
	ToFromNovRam.Teplica_set_max_fertB_time	:=	Modbus.Teplica_set_max_fertB_time;
	ToFromNovRam.Teplica_set_clear_time		:=	Modbus.Teplica_set_max_fertB_time;
	ToFromNovRam.Teplica_set_temp_pomp_cold	:=	Modbus.Teplica_set_temp_pomp_cold;
	ToFromNovRam.Teplica_set_temp_window_open	:=	Modbus.Teplica_set_temp_window_open;
	ToFromNovRam.Teplica_set_poliv_before_fert	:=	Modbus.Teplica_set_poliv_before_fert;

	ToFromNovRam.Teplica_set_temp_tank		:=	Modbus.Teplica_set_temp_tank			;
	ToFromNovRam.Teplica_fert_kf				:=	Modbus.Teplica_fert_kf				;
	ToFromNovRam.Teplica_zone_poliv			:=	Modbus.Teplica_zone_poliv			;
	ToFromNovRam.Teplica_type_fert			:=	Modbus.Teplica_type_fert				;
	ToFromNovRam.Teplica_type_poliv			:=	Modbus.Teplica_type_poliv				;
	ToFromNovRam.Teplica_set_clear_time		:=	Modbus.Teplica_set_clear_time			;
	ToFromNovRam.Teplica_set_finish_clear_time	:=	Modbus.Teplica_set_finish_clear_time;
	ToFromNovRam.Teplica_set_finish_clear_vol		:=	Modbus.Teplica_set_finish_clear_vol	;

	ToFromNovRam.Ponics_start_mintutes_poliv			:=	Modbus.Ponics_start_mintutes_poliv;
	ToFromNovRam.Ponics_start_minutes_doliv_AB		:=	Modbus.Ponics_start_minutes_doliv_AB;
	ToFromNovRam.Ponics_start_minutes_doliv_water	:=	Modbus.Ponics_start_minutes_doliv_water;
	ToFromNovRam.Ponics_set_doliv_AB				:=	Modbus.Ponics_set_doliv_AB;
	ToFromNovRam.Ponics_set_doliv_water				:=	Modbus.Ponics_set_doliv_water;
	ToFromNovRam.Ponics_set_max_poliv_time			:=	Modbus.Ponics_set_max_poliv_time;
	ToFromNovRam.Ponics_set_max_doliv_A_time		:=	Modbus.Ponics_set_max_doliv_A_time;
	ToFromNovRam.Ponics_set_max_doliv_water_time	:=	Modbus.Ponics_set_max_doliv_water_time;
	ToFromNovRam.Ponics_set_EC					:=	Modbus.Ponics_set_EC;
	ToFromNovRam.Balkon_set_temp					:=	Modbus.Balkon_set_temp;
	ToFromNovRam.Ponics_A_kf						:=	Modbus.Ponics_A_kf;
	ToFromNovRam.Ponics_B_kf						:=	Modbus.Ponics_B_kf;
	ToFromNovRam.Ponics_water_kf					:=	Modbus.Ponics_water_kf;
	ToFromNovRam.Sensor_house_water_imp			:=	Modbus.Sensor_house_water_imp;

	ToFromNovRam.Parnik_temp_step1_window			:=	Modbus.Parnik_temp_step1_window;
	ToFromNovRam.Parnik_temp_step2_window			:=	Modbus.Parnik_temp_step2_window;
	ToFromNovRam.Parnik_set_auto_window			:=	Modbus.Parnik_set_auto_window;
	ToFromNovRam.Parnik_current_level_window			:=	Modbus.Parnik_current_level_window;
	ToFromNovRam.Parnik_manual_level_window		:=	Modbus.Parnik_manual_level_window;


	teplica_new;
	ponics;
	Thermocontrol;

	Sensors;						(* Аналогвые датчики на шине KL *)
	Security_new;						(* Мониторинг датчиков охраны *)
	RS485read;					(* Опрос устройств на шине RS485 *)
	RS485read_2;					(* Опрос устройств на шине RS485 *)
(*	RS485read_3; *)					(* Опрос устройств на шине RS485 *)

(*	Mqtt;	*)					(* MQTT *)
(*	Thermocontrol; *)				(* Термостат*)
	VentControl;					(* Глобальный контроль вентустановки*)
	VentPower;					(* Авторегулировка мощности вентустановки по датчикам CO2*)
	Poliv;						(* Таймеры зонального полива *)


	Power_act;					(*Контроль резервного освещения*)
	Alarm;


(* Прямое присовение виртуальных переменных к переменным, жестко привязаным к физ. портам. Частота обновления= циклу ПЛК (50 мсек) : *)
	HW_pomp_house				:=	Modbus.Pomp_house;
	Modbus.Sensor_supply		:=	HW_sensor_supply;

	HW_kalitka					:=	Modbus.Kalitka;
	iobroker.button_light_garden	:=	HW_button_light_garden;
	HW_light_garden				:=	Modbus.Light_garden;
	iobroker.Light_garden			:=	Modbus.Light_garden;
	Modbus.Valve_status			:=	BOOL_TO_INT(HW_vent_relay_pressure);
	Modbus.Balkon_light_rassada	:=	HW_light_rassada;

	Buttons;						(*Обработка нажатия кнопок *)
	tmCheck();
	tmCheckE();
	Timer_day();
	Timer_CO2();
	tmcheckM();

	Modbus.PLC_uptime			:=	SystemTaskInfoArr[1].cycleCount;
	HW_teplica_pomp_fert_level	:=	Modbus.Teplica_pomp_fert_level;
	HW_teplica_pomp_poliv	:=	Modbus.Teplica_pomp_poliv;
	Modbus.Battery_low		:=	HW_battery_low;

(*	IF (Modbus.Teplica_pomp_fertA = TRUE OR Modbus.Teplica_pomp_fertB = TRUE) THEN
		HW_teplica_pomp_fertA	:=	TRUE;
	ELSE
				HW_teplica_pomp_fertA	:=	FALSE;
	END_IF
*)
(*	HW_teplica_zone_poliv	:=	Modbus.Teplica_zone_poliv; *)



	ParnikWindowCtrl;
	Parnik_heat;






END_IF
END_PROGRAM

(* POU teplica_new, ST *)
PROGRAM teplica_new
VAR
	Cnt_water_fertA_start	:	UDINT;
	Cnt_water_fertB_start	:	UDINT;
	Cnt_water_finish_clear_start	:	UDINT;
	Cnt_water_finish_clear	:		REAL;
	t_Started_poliv			:	TIME;
	t_Started_fertA			:	TIME;
	t_Started_fertB			:	TIME;


	Timer_poliv_all			: TON;
	Timer_poliv_allQ			: BOOL;

	Timer_1_clear			: TON;
	Timer_2_fertA				: TON;
	Timer_3_clear			: TON;
	Timer_4_fertB				: TON;
	Timer_poliv_with_fert		: TON;
	Timer_poliv_finish			: TON;

	Timer_calc_kf			: TON;
	Timer_calc_kfQ			:BOOL;
	Cnt_water_calc_kf_start		:REAL;
	Cnt_fertA_calc_kf_start		:REAL;
	Cnt_fertB_calc_kf_start		:REAL;
	Kf_calc_fertA				: REAL:=12;
	Kf_calc_fertB				: REAL:=12;
	vol_water				: REAL;
	vol_fertA					: REAL;
	vol_fertB					: REAL;

	Timer_poliv_finishQ		: BOOL;
	Timer_1_clearQ			: BOOL;
	Timer_2_fertAQ			: BOOL;
	Timer_3_clearQ			: BOOL;
	Timer_4_fertBQ			: BOOL;



	 tTimerValue_poliv_all		: TIME:=t#60s;  (* Максимальное время полива*)
	 tTimerValue_1_clear		: TIME:=t#10s;  (* Промывка перед 1 фертигацией*)
	 tTimerValue_2_fertA		: TIME:=t#30s;  (* Ограничение фертигации из бака А*)
	 tTimerValue_3_clear		: TIME:=t#60s;  (* Промывка перед OFF*)
	 tTimerValue_4_fertB		: TIME:=t#10s;  (* Ограничение фертигации из бака Б*)
	 tTimerValue_poliv_with_fert	: TIME:=t#60m;  (* Ограничение полива с фертигацией *)
	 tTimerValue_poliv_finish	: TIME:=t#3s;  (*Пауза перед статусом завршения полива для обновления регистров *)

	Timer_valve				: TON;
	Timer_valveQ			: BOOL;
	 tTimerValue_valve_water	: TIME:=t#60m;  (* Максимальное время открытия клапана подачи воды в теплицу*)

	TRIG_start_poliv			:	R_TRIG;
	TRIG_valve_tank_F		:	F_TRIG;
	TRIG_valve_tank_R		:	R_TRIG;

	TRIG_level_tank_low		:	R_TRIG;
	TRIG_level_tank_high		:	R_TRIG;

	Timer_light_avg			: TON;
	 tTimer_light_avg			: TIME:=t#1m;
	Timer_light_avgQ			: BOOL;
	Bool_poliv_before_fert		: 	BOOL;

	TRIG_poliv_break			:	R_TRIG;


	FertA_liters				:	REAL;
	FertB_liters				:	REAL;
	gisterezis_lux				:	INT:=1000;
(*	Poliv_before_fert			:	INT:=0; *)
	Timer_poliv_with_fertQ		: 	BOOL;


	max_EC					:	REAL;
	pi_fertA2 			: FB_CTRL_PI;
	pi_fertB2 			: FB_CTRL_PI;

	set_kf_fert		: INT:=12;
	start_cfg_pi_par	:BOOL;
	setA, setB, actA, actB, fOutA, fOutB	:REAL;

	avg_light_ma			: FB_CTRL_MOVING_AVERAGE;
	stParams_avg_light	: ST_CTRL_MOVING_AVERAGE_PARAMS;


	start_cfg_avg_light			:BOOL;

	avg_light					: REAL;
	arr_table					: ARRAY[1..20] OF FLOAT;
	Cnt_water_pipe			:UDINT;
	pwm_data_A	: REAL;
	pwm_cnt_A	: UDINT;
	pwm_avg_A	: REAL;
	pwm_data_B	: REAL;
	pwm_cnt_B	: UDINT;
	pwm_avg_B	: REAL;
	tank_level_low	:BOOL;
	tank_level_high	:BOOL;
	anti_hum_light	:BOOL;
(*	k_popr:	REAL; *)

END_VAR
IF NOT start_cfg_avg_light THEN

	stParams_avg_light.tCtrlCycleTime			:= T#60s;
	stParams_avg_light.tTaskCycleTime 			:= T#10ms;
	stParams_avg_light.nSamplesToFilter		:= 20;
	stParams_avg_light.pWorkArray_ADR		:= ADR(arr_table);
	stParams_avg_light.nWorkArray_SIZEOF		:= SIZEOF(arr_table);
	start_cfg_avg_light							:= TRUE;
END_IF

avg_light_ma(fIn:=Modbus.Teplica_light_lux, fManSyncValue :=0, bSync:=0, eMode:=eCTRL_MODE_ACTIVE,bHold:=0, stParams:=stParams_avg_light,  fOut =>avg_light);
Modbus.Teplica_avg_lux	:=	avg_light;


start_cfg_pi_par:=	FALSE;
IF NOT start_cfg_pi_par THEN


	pi_par_fertA.bARWOnIPartOnly:=0;
	pi_par_fertA.fKp:=300000*0.7;
	pi_par_fertA.fOutMaxLimit:=32765*0.7;
	pi_par_fertA.fOutMinLimit:=32765*0.25;

(*	pi_par_fertA.fOutMinLimit:=16800; *)
(*	pi_par_fertA.fOutMinLimit:=13100; *)
(*	pi_par_fertA.fOutMinLimit:=11460; *)
	pi_par_fertA.tCtrlCycleTime:=T#4s;
	pi_par_fertA.tTaskCycleTime:=T#10ms;
	pi_par_fertA.tTn:=T#12s;

	pi_par_fertB.bARWOnIPartOnly:=0;
	pi_par_fertB.fKp:=300000*0.7;
	pi_par_fertB.fOutMaxLimit:=32765*0.7;
	pi_par_fertB.fOutMinLimit:=32765*0.25;
(*	pi_par_fertB.fOutMinLimit:=16800; *)
(*	pi_par_fertB.fOutMinLimit:=13100; *)
(*	pi_par_fertA.fOutMinLimit:=11460; *)
	pi_par_fertB.tCtrlCycleTime:=T#4s;
	pi_par_fertB.tTaskCycleTime:=T#10ms;
	pi_par_fertB.tTn:=T#12s;

	start_cfg_pi_par			:=	TRUE;

END_IF


IF (Kf_calc_fertA = 0) THEN
	Kf_calc_fertA := Modbus.Teplica_fert_kf;
END_IF
IF (Kf_calc_fertB = 0) THEN
	Kf_calc_fertB := Modbus.Teplica_fert_kf;
END_IF
IF (Modbus.Teplica_fert_kf = 0) THEN
	Modbus.Teplica_fert_kf := 48;
END_IF

CASE Modbus.Teplica_fert_kf OF

79:
		pi_par_fertA.fOutMaxLimit:=32765*0.41*1.1;
		pi_par_fertA.fOutMinLimit:=32765*0.41*0.9;
		pi_par_fertB.fOutMaxLimit:=32765*0.42*1.05;
		pi_par_fertB.fOutMinLimit:=32765*0.42*0.95;

62:
		pi_par_fertA.fOutMaxLimit:=32765*0.5*1.1;
		pi_par_fertA.fOutMinLimit:=32765*0.5*0.8;
		pi_par_fertB.fOutMaxLimit:=32765*0.58*1.1;
		pi_par_fertB.fOutMinLimit:=32765*0.58*0.8;

49:
		pi_par_fertA.fOutMaxLimit:=32765*0.5*1.1;
		pi_par_fertA.fOutMinLimit:=32765*0.5*0.9;
		pi_par_fertB.fOutMaxLimit:=32765*0.58*1.1;
		pi_par_fertB.fOutMinLimit:=32765*0.58*0.9;

39:
		pi_par_fertA.fOutMaxLimit:=32765*0.53*1.1;
		pi_par_fertA.fOutMinLimit:=32765*0.53*0.9;
		pi_par_fertB.fOutMaxLimit:=32765*0.69*1.1;
		pi_par_fertB.fOutMinLimit:=32765*0.69*0.9;

30:
		pi_par_fertA.fOutMaxLimit:=32765*0.56*1.1;
		pi_par_fertA.fOutMinLimit:=32765*0.56*0.9;
		pi_par_fertB.fOutMaxLimit:=32765*0.73*1.1;
		pi_par_fertB.fOutMinLimit:=32765*0.73*0.9;

24:
		pi_par_fertA.fOutMaxLimit:=32765*0.6*1.1;
		pi_par_fertA.fOutMinLimit:=32765*0.6*0.9;
		pi_par_fertB.fOutMaxLimit:=32765*0.75*1.1;
		pi_par_fertB.fOutMinLimit:=32765*0.75*0.9;


END_CASE


setA		:=	1/(INT_TO_REAL(Modbus.Teplica_fert_kf));

setB		:=	1/(INT_TO_REAL(Modbus.Teplica_fert_kf));


(*
Trigger_water_impulse_teplica(CLK:=HW_impulse_water_teplica);
Trigger_fertA_impulse_teplica(CLK:=HW_impulse_fertA_teplica);
Trigger_fertB_impulse_teplica(CLK:=HW_impulse_fertB_teplica);

IF Trigger_water_impulse_teplica.Q THEN
	Modbus.Teplica_impulse_water_cnt	:= 	Modbus.Teplica_impulse_water_cnt+1;
END_IF


IF Trigger_fertA_impulse_teplica.Q THEN
	Modbus.Teplica_impulse_fertA_cnt	:= 	Modbus.Teplica_impulse_fertA_cnt+1;
END_IF
IF Trigger_fertB_impulse_teplica.Q THEN
	Modbus.Teplica_impulse_fertB_cnt	:= 	Modbus.Teplica_impulse_fertB_cnt+1;
END_IF
*)
tTimerValue_poliv_all	:=	UDINT_TO_TIME(60*1000*Modbus.Teplica_set_max_poliv_time);
tTimerValue_1_clear	:=	UDINT_TO_TIME(60*1000*Modbus.Teplica_set_clear_time);
tTimerValue_2_fertA	:=	UDINT_TO_TIME(60*1000*Modbus.Teplica_set_max_fertA_time);
tTimerValue_3_clear	:=	UDINT_TO_TIME(60*1000*Modbus.Teplica_set_finish_clear_time);
tTimerValue_4_fertB	:=	UDINT_TO_TIME(60*1000*Modbus.Teplica_set_max_fertB_time);

Timer_poliv_all();
Timer_poliv_with_fert();
Timer_1_clear();
Timer_2_fertA();
Timer_3_clear();
Timer_4_fertB();
Timer_valve();
Timer_poliv_finish();
Timer_calc_kf();

TRIG_start_poliv(CLK :=Modbus.Teplica_poliv_active);
TRIG_poliv_break(CLK :=Modbus.Teplica_poliv_break);

TRIG_valve_tank_F(CLK:=HW_water_tank_teplica_level);
TRIG_valve_tank_R(CLK:=HW_water_tank_teplica_level);

IF (Modbus.Teplica_tank_level <1000) THEN
	tank_level_low	:=	TRUE;
	tank_level_high	:=	FALSE;
END_IF
IF (Modbus.Teplica_tank_level >1200) THEN
	tank_level_high	:=	TRUE;
	tank_level_low	:=	FALSE;
END_IF



TRIG_level_tank_low(CLK:= tank_level_low);
TRIG_level_tank_high(CLK:= tank_level_high);

Modbus.Teplica_tank_teplica_level	:=	HW_water_tank_teplica_level;

IF (TRIG_valve_tank_F.Q OR TRIG_level_tank_low.Q ) THEN
	Timer_valve(IN:=NOT Timer_valveQ , PT:=tTimerValue_valve_water , Q=>Timer_valveQ , ET=> );
	HW_valve_pomp_teplica :=	TRUE;
	Modbus.Teplica_valve_water_in		:=	TRUE;
END_IF


IF (TRIG_valve_tank_R.Q	OR Timer_valveQ = TRUE OR TRIG_level_tank_high.Q) THEN
	HW_valve_pomp_teplica :=	FALSE;
	Modbus.Teplica_valve_water_in		:=	FALSE;
	Timer_valveQ	:= FALSE;
	Timer_valve.IN	:= FALSE;
END_IF



IF (TRIG_start_poliv.Q  (*AND Modbus.Teplica_tank_level > 400 *) )   THEN
		pwm_data_A	:=	0;
		pwm_cnt_A	:=	0;
		pwm_avg_A	:=	0;
		pwm_data_B	:=	0;
		pwm_cnt_B	:=	0;
		pwm_avg_B	:=	0;


		Cnt_water_pipe	:=	0;
		Poliv_liters	:=	0;
		FertA_liters	:=	0;
		FertB_liters	:=	0;
		Cnt_water_fertA_start	:=	0;
		Cnt_water_fertB_start	:=	0;
		Cnt_water_finish_clear	:=	0;
		Cnt_water_finish_clear_start		:=	0;
		Modbus.Teplica_impulse_water_cnt	:=	0;
		Modbus.Teplica_impulse_fertA_cnt	:=	0;
		Modbus.Teplica_impulse_fertB_cnt	:=	0;
		Modbus.Teplica_cnt_water_pipe			:=	0;

		Modbus.Teplica_time_elapsed_poliv :=0;
		Modbus.Teplica_time_elapsed_fertA :=0;
		Modbus.Teplica_time_elapsed_fertB :=0;
		max_EC	:=	0;
		Timer_1_clearQ			:= FALSE;
		Timer_2_fertAQ			:= FALSE;
		Timer_3_clearQ			:= FALSE;
		Timer_4_fertBQ			:= FALSE;
		Timer_poliv_finishQ		:= FALSE;
		Timer_calc_kfQ			:=FALSE;
		Bool_poliv_before_fert		:=FALSE;
		Modbus.Teplica_pomp_poliv:=TRUE;

		Timer_poliv_all.IN := FALSE;
		Timer_poliv_with_fert.IN := FALSE;
		Timer_1_clear.IN := FALSE;
		Timer_2_fertA.IN:=FALSE;
		Timer_3_clear.IN := FALSE;
		Timer_4_fertB.IN:=FALSE;
		Timer_calc_kf.IN	:=	FALSE;
		Timer_poliv_finish.IN := FALSE;

		 t_Started_poliv := TIME();
		Timer_poliv_all(IN:=NOT Timer_poliv_allQ , PT:=tTimerValue_poliv_all , Q=>Timer_poliv_allQ , ET=> );
		Timer_poliv_with_fert(IN:=NOT Timer_poliv_with_fertQ , PT:=tTimerValue_poliv_with_fert , Q=>Timer_poliv_with_fertQ , ET=> );
		Timer_1_clear(IN:=NOT Timer_1_clearQ , PT:=tTimerValue_1_clear , Q=>Timer_1_clearQ , ET=> );
		Modbus.Teplica_poliv_status_PLC:=2;
		IF  (Modbus.Teplica_zone_poliv = 0) THEN
			Modbus.Teplica_poliv_message_PLC:=1;
		ELSE
			Modbus.Teplica_poliv_message_PLC:=2;
		END_IF


END_IF

IF (Modbus.Teplica_poliv_status_PLC=2  ) THEN
	Cnt_water_pipe	:=	Modbus.Teplica_cnt_water_pipe;
	Poliv_liters 	:= 	UDINT_TO_REAL(Modbus.Teplica_impulse_water_cnt)/INT_TO_REAL(Modbus.Teplica_poliv_kf);
	FertA_liters	:=	UDINT_TO_REAL(Modbus.Teplica_impulse_fertA_cnt)/INT_TO_REAL(Modbus.Teplica_fertA_kf);
	FertB_liters	:=	UDINT_TO_REAL(Modbus.Teplica_impulse_fertB_cnt)/INT_TO_REAL(Modbus.Teplica_fertB_kf);
	Modbus.Teplica_time_elapsed_poliv :=(TIME_TO_UDINT( TIME() - t_Started_poliv))/1000;

(*	pi_fertA2(fSetpointValue:=setA, fActualValue := actA, fManSyncValue :=0, bSync:=0, eMode:=2,bHold:=0, stParams:=pi_par_fertA, fOut => );
	pi_fertB2(fSetpointValue:=setB, fActualValue :=actB, fManSyncValue :=0, bSync:=0, eMode:=2,bHold:=0, stParams:=pi_par_fertB, fOut => );
	fOutA	:=	pi_fertA2.fOut;
	fOutB	:=	pi_fertB2.fOut;
*)

	IF (Modbus.Teplica_sensor_soil_EC > max_EC) THEN
		max_EC	:=	Modbus.Teplica_sensor_soil_EC;
	END_IF

(* промывка и фертигация   OR Modbus.Teplica_set_poliv_before_fert >Poliv_liters*)

	IF (Modbus.Teplica_type_poliv = TRUE) THEN  (* Полив с фертигацией*)
		IF (NOT Timer_1_clear.Q AND Bool_poliv_before_fert	= FALSE)  THEN
			IF (Modbus.Teplica_type_fert = FALSE) THEN
				IF  (Modbus.Teplica_zone_poliv = 0) THEN
						Modbus.Teplica_poliv_message_PLC:=3;
				ELSE
						Modbus.Teplica_poliv_message_PLC:=4;
				END_IF

			ELSE
				IF  (Modbus.Teplica_zone_poliv = 0) THEN
					Modbus.Teplica_poliv_message_PLC:=5;
				ELSE
					Modbus.Teplica_poliv_message_PLC:=6;
				END_IF

			END_IF
		END_IF


		IF ((Timer_1_clear.Q OR Poliv_liters>Modbus.Teplica_set_poliv_before_fert) AND Bool_poliv_before_fert=FALSE) THEN

			Timer_1_clear.IN 		:= FALSE;
			Bool_poliv_before_fert	:= TRUE;
			IF (Modbus.Teplica_type_fert = FALSE) THEN
				 (*Fert A *)
				IF  (Modbus.Teplica_zone_poliv = 0) THEN
					Modbus.Teplica_poliv_message_PLC:=7;
				ELSE
					Modbus.Teplica_poliv_message_PLC:=8;
				END_IF

				Modbus.Teplica_pomp_fertA :=  TRUE;  (*включение насоса фертигации из бака А*)
				Timer_2_fertA(IN:=NOT Timer_2_fertAQ , PT:=tTimerValue_2_fertA , Q=>Timer_2_fertAQ , ET=> );
				t_Started_fertA := TIME();
				Cnt_water_fertA_start :=Modbus.Teplica_impulse_water_cnt;
				Cnt_water_calc_kf_start	:=Poliv_liters;
				Cnt_fertA_calc_kf_start:=FertA_liters;

				Modbus.Teplica_pomp_fertB :=  TRUE;   (*включение насоса фертигации из бака B*)

				Cnt_water_fertB_start :=Modbus.Teplica_impulse_water_cnt;
				Cnt_fertB_calc_kf_start:=FertB_liters;

			END_IF
		END_IF

		IF ( (Timer_2_fertA.Q OR FertA_liters > Modbus.Teplica_set_fertA) AND Modbus.Teplica_pomp_fertA =  TRUE) THEN
			 (*start finish clear *)
			IF  (Modbus.Teplica_zone_poliv = 0) THEN
				Modbus.Teplica_poliv_message_PLC:=11;
			ELSE
				Modbus.Teplica_poliv_message_PLC:=12;
			END_IF

			Modbus.Teplica_pomp_fertA :=  FALSE; (*отключение насоса фертигации из бака А*)
			Modbus.Teplica_time_elapsed_fertA :=(TIME_TO_UDINT( TIME() - t_Started_fertA))/1000;
			Modbus.Cnt_water_fertA	:=	Modbus.Teplica_impulse_water_cnt -Cnt_water_fertA_start;

			Modbus.Teplica_pomp_fertB :=  FALSE; (*отключение насоса фертигации из бака B*)
			Modbus.Teplica_time_elapsed_fertB :=(TIME_TO_UDINT( TIME() - t_Started_fertB))/1000;
			Modbus.Cnt_water_fertB	:=	Modbus.Teplica_impulse_water_cnt -Cnt_water_fertB_start;


			Timer_2_fertA.IN:=FALSE;
			Cnt_water_finish_clear_start		:=	Modbus.Teplica_impulse_water_cnt;
			Timer_3_clear(IN:=NOT Timer_3_clearQ , PT:=tTimerValue_3_clear , Q=>Timer_3_clearQ , ET=> );

		END_IF

		IF  (Modbus.Teplica_pomp_fertA =  TRUE) THEN
			actA		:=	1/Kf_calc_fertA;
			pi_fertA2(fSetpointValue:=setA, fActualValue := actA, fManSyncValue :=0, bSync:=0, eMode:=2,bHold:=0, stParams:=pi_par_fertA, fOut => );
			fOutA	:=	pi_fertA2.fOut;
			Modbus.Teplica_time_elapsed_fertA :=(TIME_TO_UDINT( TIME() - t_Started_fertA))/1000;
			Modbus.Cnt_water_fertA	:=	Modbus.Teplica_impulse_water_cnt -Cnt_water_fertA_start;


			actB		:=	1/Kf_calc_fertB;
			pi_fertB2(fSetpointValue:=setB, fActualValue :=actB, fManSyncValue :=0, bSync:=0, eMode:=2,bHold:=0, stParams:=pi_par_fertB, fOut => );
			fOutB	:=	pi_fertB2.fOut;
			Modbus.Teplica_time_elapsed_fertB :=(TIME_TO_UDINT( TIME() - t_Started_fertB))/1000;
			Modbus.Cnt_water_fertB	:=	Modbus.Teplica_impulse_water_cnt -Cnt_water_fertB_start;

			Timer_calc_kf(IN:=NOT Timer_calc_kfQ , PT:=t#4s , Q=>Timer_calc_kfQ , ET=> );

			IF (Timer_calc_kf.Q)	THEN
			(*	vol_water	:=	Poliv_liters-Cnt_water_calc_kf_start *);
				vol_water	:=	0.46666;
				vol_fertA		:=	FertA_liters-Cnt_fertA_calc_kf_start;
				vol_fertB		:=	FertB_liters-Cnt_fertB_calc_kf_start;

				IF (vol_fertA > 0 ) THEN
					Kf_calc_fertA	:= 	 vol_water/vol_fertA;
				ELSE
					Kf_calc_fertA	:=	Modbus.Teplica_fert_kf;
				END_IF

				IF (vol_fertB > 0 ) THEN
					Kf_calc_fertB	:= 	 vol_water/vol_fertB;
				ELSE
					Kf_calc_fertB	:=	Modbus.Teplica_fert_kf;
				END_IF

				Cnt_water_calc_kf_start	:=Poliv_liters;
				Cnt_fertA_calc_kf_start:=FertA_liters;
				Cnt_fertB_calc_kf_start:=FertB_liters;

				Timer_calc_kfQ	:=	FALSE;
				Timer_calc_kf.IN	:=	FALSE;


			END_IF

			fert_pwm_levelA	:=	 REAL_TO_UINT(fOutA);
			pwm_data_A		:=	pwm_data_A + fert_pwm_levelA;
			pwm_cnt_A		:=	pwm_cnt_A + 1;
			pwm_avg_A		:=	pwm_data_A / pwm_cnt_A;

			fert_pwm_levelB	:=	 REAL_TO_UINT(fOutB);
			pwm_data_B		:=	pwm_data_B + fert_pwm_levelB;
			pwm_cnt_B		:=	pwm_cnt_B + 1;
			pwm_avg_B		:=	pwm_data_B / pwm_cnt_B;


		ELSE
			fert_pwm_levelA	:=	0;
			fert_pwm_levelB	:=	0;

		END_IF





		IF (Modbus.Teplica_poliv_message_PLC =11 OR Modbus.Teplica_poliv_message_PLC = 12 OR Modbus.Teplica_poliv_message_PLC = 13  OR Modbus.Teplica_poliv_message_PLC = 14) THEN
			Cnt_water_finish_clear	:=	UDINT_TO_REAL(Modbus.Teplica_impulse_water_cnt-Cnt_water_finish_clear_start)/Modbus.Teplica_poliv_kf;
		END_IF


		IF (Timer_poliv_with_fert.Q=TRUE OR   Modbus.Teplica_poliv_break=TRUE OR Timer_3_clear.Q=TRUE OR Cnt_water_finish_clear > Modbus.Teplica_set_finish_clear_vol  )THEN


			Modbus.Teplica_max_EC		:=	max_EC;

			Modbus.Teplica_poliv_active:= FALSE;
			Modbus.Teplica_pomp_poliv:=FALSE;
			Modbus.Teplica_pomp_fertA :=  FALSE;
			Modbus.Teplica_pomp_fertB :=  FALSE;
			Timer_poliv_all.IN := FALSE;
			Timer_poliv_with_fert.IN := FALSE;
			Timer_1_clear.IN := FALSE;
			Timer_2_fertA.IN:=FALSE;
			Timer_3_clear.IN := FALSE;
			Timer_4_fertB.IN:=FALSE;
			Timer_calc_kf.IN	:=	FALSE;
			Timer_1_clearQ			:= FALSE;
			Timer_2_fertAQ			:= FALSE;
			Timer_3_clearQ			:= FALSE;
			Timer_4_fertBQ			:= FALSE;

			IF (Modbus.Teplica_type_fert = FALSE) THEN
				 (*finished poliv with fert A*)
				IF  (Modbus.Teplica_zone_poliv = 0) THEN
					Modbus.Teplica_poliv_message_PLC:=15;
				ELSE
					Modbus.Teplica_poliv_message_PLC:=16;
				END_IF

			ELSE
				IF  (Modbus.Teplica_zone_poliv = 0) THEN
					Modbus.Teplica_poliv_message_PLC:=17;
				ELSE
					Modbus.Teplica_poliv_message_PLC:=18;
				END_IF

			END_IF

			Modbus.Teplica_poliv_status_PLC :=  10;
			Timer_poliv_finish(IN:=NOT Timer_poliv_finishQ, PT:=tTimerValue_poliv_finish , Q=>Timer_poliv_finishQ , ET=> );
		END_IF
		ELSE
			fert_pwm_levelA:=0;
			fert_pwm_levelB:=0;
	END_IF

	IF (Modbus.Teplica_type_poliv = FALSE) THEN (*Полив без фертигации*)
		IF (Timer_poliv_all.Q=TRUE OR (Poliv_liters > Modbus.Teplica_set_poliv)  OR Modbus.Teplica_poliv_break=TRUE   )THEN
			(*finished only poliv *)
			IF  (Modbus.Teplica_zone_poliv = 0) THEN
					Modbus.Teplica_poliv_message_PLC:=19;
			ELSE
					Modbus.Teplica_poliv_message_PLC:=20;
			END_IF

			Modbus.Teplica_poliv_active:= FALSE;
			Modbus.Teplica_pomp_poliv:=FALSE;
			Modbus.Teplica_pomp_fertA :=  FALSE;
			Modbus.Teplica_pomp_fertB :=  FALSE;
			Timer_poliv_all.IN := FALSE;
			Timer_poliv_with_fert.IN := FALSE;
			Timer_1_clear.IN := FALSE;
			Timer_2_fertA.IN:=FALSE;
			Timer_3_clear.IN := FALSE;
			Timer_4_fertB.IN:=FALSE;
			Timer_1_clearQ			:= FALSE;
			Timer_2_fertAQ			:= FALSE;
			Timer_3_clearQ			:= FALSE;
			Timer_4_fertBQ			:= FALSE;
			Modbus.Teplica_poliv_status_PLC :=  10;
		END_IF
	END_IF
	ELSE
		fert_pwm_levelA:=0;
		fert_pwm_levelB:=0;
END_IF

Modbus.Teplica_fert_actA			:=	Kf_calc_fertA;
Modbus.Teplica_fert_actB			:=	Kf_calc_fertB;
Modbus.Teplica_fert_pwm_levelA	:=	REAL_TO_INT(100*fert_pwm_levelA/32765);
Modbus.Teplica_fert_pwm_levelB	:=	REAL_TO_INT(100*fert_pwm_levelB/32765);
Modbus.Teplica_pwm_avg_A		:=	REAL_TO_INT(100*pwm_avg_A/32765);
Modbus.Teplica_pwm_avg_B		:=	REAL_TO_INT(100*pwm_avg_B/32765);









(*LIGHT TEPLICA *)

IF (Modbus.Teplica_light = FALSE OR anti_hum_light = TRUE) THEN

(*	IF ((Modbus.Teplica_avg_lux > Modbus.Teplica_light_set_low+gisterezis_lux OR Modbus.Teplica_temp_air>25) OR Modbus.Teplica_light_allow = FALSE  ) THEN
		Modbus.Teplica_light :=FALSE;
		HW_teplica_light		:=	FALSE;
	END_IF
*)
	IF ((Modbus.Teplica_avg_lux <  Modbus.Teplica_light_set_low-gisterezis_lux  AND Modbus.Teplica_temp_air<27) AND Modbus.Teplica_light_allow ) THEN
		Modbus.Teplica_light:=TRUE;
		HW_teplica_light		:=	TRUE;
	END_IF

	IF anti_hum_light = TRUE THEN
		Modbus.Teplica_light:=TRUE;
		HW_teplica_light		:=	TRUE;
	END_IF

END_IF

IF (Modbus.Teplica_light = TRUE AND anti_hum_light = FALSE ) THEN

	IF ((Modbus.Teplica_avg_lux  >  Modbus.Teplica_light_set_low+gisterezis_lux  OR Modbus.Teplica_temp_air>28) OR Modbus.Teplica_light_allow = FALSE  ) THEN
		Modbus.Teplica_light :=FALSE;
		HW_teplica_light		:=	FALSE;
	END_IF


END_IF



(*HEAT TEPLICA *)

	IF ((Modbus.Teplica_temp_air > Modbus.Teplica_temp_set_low+1) ) THEN
		Modbus.Teplica_heat :=FALSE;
		HW_teplica_heat		:= FALSE;
	END_IF

	IF ((Modbus.Teplica_temp_air <  Modbus.Teplica_temp_set_low-1 ) ) THEN
		Modbus.Teplica_heat:=TRUE;
		HW_teplica_heat		:=	TRUE;
	END_IF


(*HEAT TANK TEPLICA *)

	IF ((Modbus.Teplica_temp_water_tank > Modbus.Teplica_set_temp_tank+1)  OR HW_teplica_heat = TRUE  OR HW_water_tank_teplica_level = FALSE  (* OR Modbus.Teplica_tank_level < 400 *) ) THEN
		Modbus.Teplica_tank_heat :=FALSE;
	(*	HW_teplica_tank_heat		:= FALSE; *)
	END_IF

	IF ((Modbus.Teplica_temp_water_tank <  Modbus.Teplica_set_temp_tank-1 ) AND HW_teplica_heat = FALSE  AND HW_water_tank_teplica_level = TRUE  (*AND Modbus.Teplica_tank_level > 400 *)) THEN
		Modbus.Teplica_tank_heat:=TRUE;
	(*	HW_teplica_tank_heat		:=	TRUE; *)
	END_IF




(*VENT  TEPLICA *)

(* 1. КРИТИЧЕСКИЙ ХОЛОД: Если внутри ниже +12, выключаем всё принудительно *)
IF (Modbus.Teplica_temp_air < 12) THEN
    Modbus.Teplica_vent := FALSE;
    HW_teplica_vent     := FALSE;
    anti_hum_light      := FALSE;

(* 2. НОЧНОЙ РЕЖИМ (ВЛАЖНОСТЬ) С ГИСТЕРЕЗИСОМ: *)
(* Включаем свет при >85%. Но если он УЖЕ горит, то держим его включенным, пока влажность выше 80% *)
ELSIF (Modbus.Teplica_hum_SHT30 > 85) OR (anti_hum_light AND (Modbus.Teplica_hum_SHT30 > 80)) THEN
    anti_hum_light      := TRUE;  (* Включаем/держим 2кВт LED для сушки *)
    Modbus.Teplica_vent := FALSE; (* Вытяжка принудительно выключена *)
    HW_teplica_vent     := FALSE;

(* 3. ШТАТНЫЙ РЕЖИМ: Если влажность упала ниже 80% *)
ELSE
    anti_hum_light      := FALSE; (* Выключаем свет сушки *)
    
    (* Четкий гистерезис вентиляции по температуре *)
    IF (Modbus.Teplica_temp_air < Modbus.Teplica_temp_set_high - 1) THEN
        Modbus.Teplica_vent := FALSE;
        HW_teplica_vent     := FALSE;
        
    ELSIF (Modbus.Teplica_temp_air > Modbus.Teplica_temp_set_high + 1) THEN
        Modbus.Teplica_vent := TRUE;
        HW_teplica_vent     := TRUE;
    END_IF
END_IF



	IF (Modbus.Teplica_temp_air < Modbus.Teplica_set_temp_window_open-1 ) THEN
	(*	HW_teplica_window_opener		:=FALSE; *)
		Modbus.Teplica_window_opener	:=FALSE;
	END_IF
	IF (Modbus.Teplica_temp_air >  Modbus.Teplica_set_temp_window_open+1 AND   Modbus.Street_temp > 0 ) THEN
	(*	HW_teplica_window_opener		:=TRUE; *)
		Modbus.Teplica_window_opener	:=TRUE;
	END_IF


	IF (Modbus.Teplica_temp_air < Modbus.Teplica_set_temp_pomp_cold-1  OR Modbus.Street_hum >71  ) THEN
	(*	HW_teplica_pomp_cold		:=FALSE; *)
		Modbus.Teplica_pomp_cold	:=FALSE;
	END_IF
	IF (Modbus.Teplica_temp_air >  Modbus.Teplica_set_temp_pomp_cold+1 AND   Modbus.Street_temp >10  AND Modbus.Street_hum <  69) THEN
	(*	HW_teplica_pomp_cold		:=TRUE; *)
		Modbus.Teplica_pomp_cold	:=TRUE;
	END_IF
END_PROGRAM

(* POU ponics, ST *)
PROGRAM ponics
VAR

	t_Started_poliv			:	TIME;
	t_Started_AB				:	TIME;


	Timer_poliv				: TON;
	Timer_polivQ			: BOOL;

	Timer_doliv_water			: TON;
	Timer_doliv_AB			: TON;


	Timer_doliv_waterQ		: BOOL;


	 tTimerValue_poliv		: TIME:=t#60s;  (* Максимальное время полива*)
	 tTimerValue_doliv_water	: TIME:=t#10s;  (* Промывка перед 1 фертигацией*)
	 tTimerValue_doliv_AB		: TIME:=t#30s;

	Timer_doliv_ABQ			:	BOOL;
	TRIG_start_poliv			:	R_TRIG;
	TRIG_start_doliv_water		:	R_TRIG;
	TRIG_start_doliv_AB		:	R_TRIG;
	TRIG_poliv_break			:	R_TRIG;

	Doliv_liters				:	REAL;
	Doliv_liters_int			:	REAL;
	Tank_A_liters				:	REAL;
	Tank_B_liters				:	REAL;
	gisterezis_lux				:	INT:=1000;
(*
	Trigger_water_impulse_ponics	: F_TRIG;
	Trigger_A_impulse_ponics		: F_TRIG;
	Trigger_B_impulse_ponics		: F_TRIG;
*)

	TRIG_valve_tank_F		:	F_TRIG;
	TRIG_valve_tank_R		:	R_TRIG;
	PLC_status				:	BYTE;

	Ponics_poliv_start			:	TOD;
	Ponics_poliv_end			:	TOD;
	Ponics_doliv_AB_start			:	TOD;
	Ponics_doliv_AB_end			:	TOD;
	Ponics_doliv_water_start			:	TOD;
	Ponics_doliv_water_end			:	TOD;
	Ponics_light_morning_start			:	TOD;
	Ponics_light_morning_end			:	TOD;
	dtCurrentDate         		: DT;
	fileTime              		: T_FILETIME;
	fbGetSystemTime       	: GETSYSTEMTIME;
	time_now			: TOD;
	tz					: TIME:=T#5h;
	test1, test2, test3 ,hours,minutes		: INT;
	hm				:ExtractTime;
	Ponics_impulse_water_cnt_int	:UDINT;
	Timer_block_dolivAB			:TON;
	Timer_block_dolivABQ			:BOOL;
	Timer_block_doliv_water			:TON;
	Timer_block_doliv_waterQ			:BOOL;

	t_Started_doliv_A			:	TIME;
	t_Started_doliv_B			:	TIME;
	t_Started_doliv_water		:	TIME;

	pi_balkon 			: FB_CTRL_PI;
	pwm_balkon			: FB_CTRL_PWM_OUT;

END_VAR
tTimerValue_poliv			:=	UDINT_TO_TIME(1000*Modbus.Ponics_set_max_poliv_time);
tTimerValue_doliv_water	:=	UDINT_TO_TIME(1000*Modbus.Ponics_set_max_doliv_water_time);
tTimerValue_doliv_AB		:=	UDINT_TO_TIME(1000*Modbus.Ponics_set_max_doliv_A_time);

Timer_poliv();
Timer_doliv_water();
Timer_doliv_AB();
Timer_block_dolivAB();
Timer_block_doliv_water();

fbGetSystemTime(timeLoDW =>fileTime.dwLowDateTime,
                timeHiDW =>fileTime.dwHighDateTime);
dtCurrentDate:=FILETIME_TO_DT(fileTime);
time_now	:= DT_TO_TOD(dtCurrentDate)+tz;

Ponics_poliv_start					:=	UDINT_TO_TOD(Modbus.Ponics_poliv_start);
Ponics_poliv_end					:=	UDINT_TO_TOD(Modbus.Ponics_poliv_end);
Ponics_doliv_AB_start				:=	UDINT_TO_TOD(Modbus.Ponics_doliv_AB_start);
Ponics_doliv_AB_end				:=	UDINT_TO_TOD(Modbus.Ponics_doliv_AB_end);
Ponics_doliv_water_start			:=	UDINT_TO_TOD(Modbus.Ponics_doliv_water_start);
Ponics_doliv_water_end			:=	UDINT_TO_TOD(Modbus.Ponics_doliv_water_end);
Ponics_light_morning_start			:=	UDINT_TO_TOD(Modbus.Ponics_light_morning_start);
Ponics_light_morning_end			:=	UDINT_TO_TOD(Modbus.Ponics_light_morning_end);

hm(tm:=time_now, h=>hours, m=>minutes);

IF (time_now>Ponics_poliv_start AND time_now<Ponics_poliv_end AND minutes =  Modbus.Ponics_start_mintutes_poliv AND HW_Ponics_pomp_main =	FALSE ) THEN
	Modbus.Ponics_poliv_active	:= TRUE;
END_IF

IF  ( Modbus.Ponics_doliv_AB_active	= FALSE AND time_now>Ponics_doliv_AB_start AND time_now<Ponics_doliv_AB_end AND minutes =  Modbus.Ponics_start_minutes_doliv_AB AND HW_Ponics_pomp_tankA =	FALSE AND HW_Ponics_pomp_tankB =	FALSE)  THEN
	Modbus.Ponics_doliv_AB_active	:= TRUE;
	Timer_block_dolivAB(IN:=NOT Timer_block_dolivABQ , PT:=T#70s , Q=>Timer_block_dolivABQ , ET=> );
END_IF

IF Timer_block_dolivAB.Q THEN
	Timer_block_dolivAB.IN			:= FALSE;
	Modbus.Ponics_doliv_AB_active	:= FALSE;
	Timer_block_dolivABQ				:= FALSE;
END_IF

IF (Modbus.Ponics_doliv_water_active	= FALSE AND time_now>Ponics_doliv_water_start AND time_now<Ponics_doliv_water_end AND minutes =  Modbus.Ponics_start_minutes_doliv_water AND HW_Ponics_pomp_water =	FALSE ) THEN
	Modbus.Ponics_doliv_water_active	:= TRUE;
	Timer_block_doliv_water(IN:=NOT Timer_block_doliv_waterQ , PT:=T#70s , Q=>Timer_block_doliv_waterQ , ET=> );
END_IF

IF Timer_block_doliv_water.Q THEN
	Timer_block_doliv_water.IN			:= FALSE;
	Modbus.Ponics_doliv_water_active	:= FALSE;
	Timer_block_doliv_waterQ			:= FALSE;
END_IF

(*
Trigger_water_impulse_ponics(CLK:=HW_impulse_water_ponics);
Trigger_A_impulse_Ponics(CLK:=HW_impulse_tankA_Ponics);
Trigger_B_impulse_Ponics(CLK:=HW_impulse_tankB_Ponics);


IF Trigger_water_impulse_Ponics.Q THEN
	Modbus.Ponics_impulse_water_cnt	:= 	Modbus.Ponics_impulse_water_cnt+1;
END_IF
IF Trigger_A_impulse_Ponics.Q THEN
	Modbus.Ponics_impulse_A_cnt	:= 	Modbus.Ponics_impulse_A_cnt+1;
END_IF
IF Trigger_B_impulse_Ponics.Q THEN
	Modbus.Ponics_impulse_B_cnt	:= 	Modbus.Ponics_impulse_B_cnt+1;
END_IF
*)

TRIG_start_poliv(CLK :=Modbus.Ponics_poliv_active);
Modbus.Ponics_poliv_active	:=	FALSE;

TRIG_poliv_break(CLK :=Modbus.Ponics_poliv_break);
TRIG_start_doliv_AB(CLK :=Modbus.Ponics_doliv_AB_active);
TRIG_start_doliv_water(CLK :=Modbus.Ponics_doliv_water_active);


(* poliv *)

IF (TRIG_start_poliv.Q AND HW_sensor_fluid_alarm = FALSE )   THEN
		Modbus.Ponics_time_elapsed_poliv :=0;
		Timer_polivQ					:= FALSE;
		Modbus.Ponics_pomp_poliv	:= TRUE;
		HW_Ponics_pomp_main		:= TRUE;
		 t_Started_poliv				:= TIME();
		Timer_poliv(IN:=NOT Timer_polivQ , PT:=tTimerValue_poliv , Q=>Timer_polivQ , ET=> );
		PLC_status.0					:= 1;
END_IF

IF ( Timer_poliv.Q OR Modbus.Ponics_poliv_break=TRUE ) THEN
		Timer_poliv.IN				:= FALSE;
		Timer_polivQ					:= FALSE;
		Modbus.Ponics_pomp_poliv	:= FALSE;
		HW_Ponics_pomp_main		:= FALSE;
		PLC_status.0					:= 0;
END_IF

TRIG_valve_tank_F(CLK:=HW_water_tank_Ponics_level_low);
TRIG_valve_tank_R(CLK:=HW_water_tank_Ponics_level_low);
Modbus.Ponics_tank_water_level	:=	HW_water_tank_Ponics_level_low;
Modbus.Ponics_tank_water_level_high	:=	HW_water_tank_Ponics_level_high;

IF (HW_Ponics_pomp_water = TRUE) THEN
	Doliv_liters 								:= UDINT_TO_REAL(Modbus.Ponics_impulse_water_cnt)/UINT_TO_REAL(Modbus.Ponics_water_kf);
	Doliv_liters_int 							:= UDINT_TO_REAL(Ponics_impulse_water_cnt_int)/UINT_TO_REAL(Modbus.Ponics_water_kf);
	Modbus.Ponics_time_elapsed_doliv_water	:= (TIME_TO_UDINT( TIME() - t_Started_doliv_water))/1000;
END_IF

IF (HW_Ponics_pomp_tankA = TRUE) THEN
	Tank_A_liters								:= UDINT_TO_REAL(Modbus.Ponics_impulse_A_cnt)/UINT_TO_REAL(Modbus.Ponics_A_kf);
	Modbus.Ponics_time_elapsed_doliv_A		:= (TIME_TO_UDINT( TIME() - t_Started_doliv_A))/1000;
END_IF

IF (HW_Ponics_pomp_tankB = TRUE) THEN
	Tank_B_liters								:= UDINT_TO_REAL(Modbus.Ponics_impulse_B_cnt)/UINT_TO_REAL(Modbus.Ponics_B_kf);
	Modbus.Ponics_time_elapsed_doliv_B		:= (TIME_TO_UDINT( TIME() - t_Started_doliv_B))/1000;
END_IF

(*  doliv water schedule if EC up  OR lelel in tank is low    *)

(*start doliv water *)
 IF (TRIG_start_doliv_water.Q    AND  HW_water_tank_Ponics_level_high = TRUE  AND HW_sensor_fluid_alarm = FALSE  AND (HW_water_tank_Ponics_level_low = TRUE OR  Modbus.Ponics_EC >  Modbus.Ponics_set_EC*1.1)   )   THEN
		Modbus.Ponics_impulse_water_cnt	:=	0;
		Doliv_liters						:=	0;
		HW_Ponics_pomp_water			:=	TRUE;
		Modbus.Ponics_pomp_doliv_water	:=	TRUE;
		t_Started_doliv_water				:=	TIME();
		Timer_doliv_water(IN:=NOT Timer_doliv_waterQ , PT:=tTimerValue_doliv_water , Q=>Timer_doliv_waterQ , ET=> );
		PLC_status.1						:=	1;
END_IF

(* stop doliv water*)

IF ( HW_Ponics_pomp_water = TRUE AND (   HW_water_tank_Ponics_level_high = FALSE	 OR Doliv_liters >Modbus. Ponics_set_doliv_water  ) 	) THEN
		Modbus.Ponics_pomp_doliv_water	:=	FALSE;
		HW_Ponics_pomp_water			:=	FALSE;
		Timer_block_doliv_water.IN			:= FALSE;
		Modbus.Ponics_doliv_water_active	:= FALSE;
		PLC_status.1						:=	0;
END_IF


IF ( Timer_doliv_water.Q  ) THEN
		Timer_doliv_water.IN				:=	FALSE;
		Timer_doliv_waterQ				:=	FALSE;
		Modbus.Ponics_pomp_doliv_water	:=	FALSE;
		HW_Ponics_pomp_water			:=	FALSE;
		PLC_status.1						:=	0;
END_IF


(*  doliv tank A, B  if EC down*)
(* (TRIG_start_doliv_AB.Q AND Modbus.Ponics_EC < Modbus.Ponics_set_EC )*) (* AND HW_water_tank_Ponics_level_high = TRUE *)
IF (TRIG_start_doliv_AB.Q   AND Modbus.Ponics_EC < Modbus.Ponics_set_EC*0.98  AND HW_sensor_fluid_alarm = FALSE)   THEN
		Modbus.Ponics_impulse_A_cnt	:=	0;
		Modbus.Ponics_impulse_B_cnt	:=	0;
		Tank_A_liters					:=	0;
		Tank_B_liters					:=	0;
		Modbus.Ponics_pomp_doliv_A	:=	TRUE;
		HW_Ponics_pomp_tankA		:=	TRUE;
		Modbus.Ponics_pomp_doliv_B	:=	TRUE;
		HW_Ponics_pomp_tankB		:=	TRUE;
		t_Started_AB					 :=	 TIME();
		t_Started_doliv_A				:=	TIME();
		t_Started_doliv_B				:=	TIME();
		Timer_doliv_AB(IN:=NOT Timer_doliv_ABQ , PT:=tTimerValue_doliv_AB , Q=>Timer_doliv_ABQ , ET=> );
		PLC_status.2					:=	1;
		PLC_status.3					:=	1;
		PLC_status.4					:=	1;
END_IF

IF ( Tank_A_liters >Modbus. Ponics_set_doliv_AB ) THEN
		Modbus.Ponics_pomp_doliv_A		:=	FALSE;
		HW_Ponics_pomp_tankA			:=	FALSE;
		PLC_status.2						:=	0;
END_IF


IF (  Tank_B_liters >Modbus. Ponics_set_doliv_AB ) THEN
		Modbus.Ponics_pomp_doliv_B		:=	FALSE;
		HW_Ponics_pomp_tankB			:=	FALSE;
		PLC_status.3						:=	0;
END_IF

IF ( Timer_doliv_AB.Q  ) THEN
		Timer_doliv_AB.IN				:=	FALSE;
		Timer_doliv_ABQ					:=	FALSE;
		Modbus.Ponics_pomp_doliv_A		:=	FALSE;
		HW_Ponics_pomp_tankA			:=	FALSE;
		Modbus.Ponics_pomp_doliv_B		:=	FALSE;
		HW_Ponics_pomp_tankB			:=	FALSE;
		PLC_status.2						:=	0;
		PLC_status.3						:=	0;
		PLC_status.4						:=	0;
END_IF


IF ( HW_sensor_fluid_alarm = TRUE  ) THEN
		Timer_poliv.IN					:=	FALSE;
		Timer_polivQ						:=	FALSE;
		Modbus.Ponics_pomp_poliv		:=	FALSE;
		HW_Ponics_pomp_main			:=	FALSE;
		PLC_status.0						:=	0;
		Timer_doliv_water.IN				:=	FALSE;
		Timer_doliv_waterQ				:=	FALSE;
		Modbus.Ponics_pomp_doliv_water	:=	FALSE;
		HW_Ponics_pomp_water			:=	FALSE;
		PLC_status.1						:=	0;
		Timer_doliv_AB.IN				:=	FALSE;
		Timer_doliv_ABQ					:=	FALSE;
		Modbus.Ponics_pomp_doliv_A		:=	FALSE;
		HW_Ponics_pomp_tankA			:=	FALSE;
		Modbus.Ponics_pomp_doliv_B		:=	FALSE;
		HW_Ponics_pomp_tankB			:=	FALSE;
		PLC_status.2						:=	0;
		PLC_status.3						:=	0;
		PLC_status.4						:=	0;
END_IF




Modbus.Ponics_status_PLC:=PLC_status;


(*LIGHT Ponics *)
IF (time_now>Ponics_light_morning_start AND time_now<Ponics_light_morning_end  ) THEN
	HW_light_rassada		:=	TRUE;
	Modbus.Balkon_set_temp	:=	Modbus.Balkon_set_temp_day;
ELSE
	HW_light_rassada		:=	FALSE;
	Modbus.Balkon_set_temp	:=	Modbus.Balkon_set_temp_night;
END_IF

Modbus.Balkon_light_rassada	:=	HW_light_rassada;



(*HEAT Ponics *)
(*
	IF ((Modbus.Balkon_temp > Modbus.Balkon_set_temp+1)   ) THEN
		HW_balkon_heat		:= FALSE;
	END_IF

	IF ((Modbus.Balkon_temp <  Modbus.Balkon_set_temp-1 ) ) THEN
		HW_balkon_heat		:=	TRUE;
	END_IF
*)
(*
pwm_par_balkon.bInstantPWMUpdate:=0;
pwm_par_balkon.tPWMPeriod:=T#5800ms;
pwm_par_balkon.tTaskCycleTime:=T#5ms;

